Fanuc TP program (LS listing): GST_CLAMSHELL_L1.LS

/PROG  GST_CLAMSHELL_L1
/ATTR
OWNER           = MNEDITOR;
COMMENT         = "BY ROBOTMASTER";
PROG_SIZE       = 0;
CREATE          = DATE 23-01-04  TIME 08:18:11;
MODIFIED        = DATE 23-01-04  TIME 08:18:11;
FILE_NAME       = ;
VERSION         = 0;
LINE_COUNT      = 5014;
MEMORY_SIZE     = 0;
PROTECT         = READ_WRITE;
TCD:  STACK_SIZE        = 0,
      TASK_PRIORITY     = 50,
      TIME_SLICE        = 0,
      BUSY_LAMP_OFF     = 0,
      ABORT_REQUEST     = 0,
      PAUSE_REQUEST     = 0;
DEFAULT_GROUP   = 1,*,*,*,*;
CONTROL_CODE = 00000000 00000000;
/MN
   1: ;
   2: ! Home ;
   3: ;
   4:  UFRAME_NUM = 7 ;
   5:  UTOOL_NUM = 3 ;
   6: ! Jump to specified pass ;
   7: R[215:passLbl] = 100 + R[180:j];
   8: ! Specify last pass ;
   9: IF R[180:j]>1,JMP LBL[8999] ;
  10: IF R[180:j]>0,JMP LBL[R[215:passLbl]] ;
  11:J P[1]  R[225] % FINE ;
  12: ;
  13: ! Path ;
  14: ;
  15:J P[2]  R[225] % FINE ;
  16:L P[3]  R[157] mm/sec CNT100 Offset,PR[24:Rotate_Offset] ;
  17:L P[4]  R[157] mm/sec CNT100 Offset,PR[24:Rotate_Offset] ;
  18: !Pass1 ;
  19: LBL[101:Pass1] ;
  20:L P[5]  R[157] mm/sec FINE Offset,PR[78:Offst_apprch]  ;
  21: WAIT   0.20(sec) ;
  22:L P[5]  R[157] mm/sec CNT100 TA    0.00sec,CALL RUN_LASER_START Offset,PR[25:Start_Offset] ;
  24:L P[6]  R[157] mm/sec CNT100 Offset,PR[24:Rotate_Offset] ;
  25:L P[7]  R[157] mm/sec CNT100 Offset,PR[24:Rotate_Offset] ;
  26:L P[8]  R[157] mm/sec CNT100 Offset,PR[24:Rotate_Offset] ;
  27:L P[9]  R[157] mm/sec CNT100 Offset,PR[24:Rotate_Offset] ;
  28:L P[10]  R[157] mm/sec CNT100 Offset,PR[24:Rotate_Offset] ;
  29:L P[11]  R[157] mm/sec CNT100 Offset,PR[24:Rotate_Offset] ;
  30:L P[12]  R[157] mm/sec CNT100 Offset,PR[24:Rotate_Offset] ;
  31:L P[13]  R[157] mm/sec CNT100 Offset,PR[24:Rotate_Offset] ;
  32:L P[14]  R[157] mm/sec CNT100 Offset,PR[24:Rotate_Offset] ;
  33:L P[15]  R[157] mm/sec CNT100 Offset,PR[24:Rotate_Offset] ;
  34:L P[16]  R[157] mm/sec CNT100 Offset,PR[24:Rotate_Offset] ;
  35:L P[17]  R[157] mm/sec CNT100 Offset,PR[24:Rotate_Offset] ;
  36:L P[18]  R[157] mm/sec CNT100 Offset,PR[24:Rotate_Offset] ;
  37:L P[19]  R[157] mm/sec CNT100 Offset,PR[24:Rotate_Offset] ;
  38:L P[20]  R[157] mm/sec CNT100 Offset,PR[24:Rotate_Offset] ;
  39:L P[21]  R[157] mm/sec CNT100 Offset,PR[24:Rotate_Offset] ;
  40:L P[22]  R[157] mm/sec CNT100 Offset,PR[24:Rotate_Offset] ;
  41:L P[23]  R[157] mm/sec CNT100 Offset,PR[24:Rotate_Offset] ;
  42:L P[24]  R[157] mm/sec CNT100 Offset,PR[24:Rotate_Offset] ;
  43:L P[25]  R[157] mm/sec CNT100 Offset,PR[24:Rotate_Offset] ;
  44:L P[26]  R[157] mm/sec CNT100 Offset,PR[24:Rotate_Offset] ;
  45:L P[27]  R[157] mm/sec CNT100 Offset,PR[24:Rotate_Offset] ;
  46:L P[28]  R[157] mm/sec CNT100 Offset,PR[24:Rotate_Offset] ;
  47:L P[29]  R[157] mm/sec CNT100 Offset,PR[24:Rotate_Offset] ;
  48:L P[30]  R[157] mm/sec CNT100 Offset,PR[24:Rotate_Offset] ;
  49:L P[31]  R[157] mm/sec CNT100 Offset,PR[24:Rotate_Offset] ;
  50:L P[32]  R[157] mm/sec CNT100 Offset,PR[24:Rotate_Offset] ;
  51:L P[33]  R[157] mm/sec CNT100 Offset,PR[24:Rotate_Offset] ;
  52:L P[34]  R[157] mm/sec CNT100 Offset,PR[24:Rotate_Offset] ;
  53:L P[35]  R[157] mm/sec CNT100 Offset,PR[24:Rotate_Offset] ;
  54:L P[36]  R[157] mm/sec CNT100 Offset,PR[24:Rotate_Offset] ;
  55:L P[37]  R[157] mm/sec CNT100 Offset,PR[24:Rotate_Offset] ;
  56:L P[38]  R[157] mm/sec CNT100 Offset,PR[24:Rotate_Offset] ;
  57:L P[39]  R[157] mm/sec CNT100 Offset,PR[24:Rotate_Offset] ;
  58:L P[40]  R[157] mm/sec CNT100 Offset,PR[24:Rotate_Offset] ;
  59:L P[41]  R[157] mm/sec CNT100 Offset,PR[24:Rotate_Offset] ;
  60:L P[42]  R[157] mm/sec CNT100 Offset,PR[24:Rotate_Offset] ;
  61:L P[43]  R[157] mm/sec CNT100 Offset,PR[24:Rotate_Offset] ;
  62:L P[44]  R[157] mm/sec CNT100 Offset,PR[24:Rotate_Offset] ;
  63:L P[45]  R[157] mm/sec CNT100 Offset,PR[24:Rotate_Offset] ;
  64:L P[46]  R[157] mm/sec CNT100 Offset,PR[24:Rotate_Offset] ;
  65:L P[47]  R[157] mm/sec CNT100 Offset,PR[24:Rotate_Offset] ;
  66:L P[48]  R[157] mm/sec CNT100 Offset,PR[24:Rotate_Offset] ;
  67:L P[49]  R[157] mm/sec CNT100 Offset,PR[24:Rotate_Offset] ;
  68:L P[50]  R[157] mm/sec CNT100 Offset,PR[24:Rotate_Offset] ;
  69:L P[51]  R[157] mm/sec CNT100 Offset,PR[24:Rotate_Offset] ;
  70:L P[52]  R[157] mm/sec CNT100 Offset,PR[24:Rotate_Offset] ;
  71:L P[53]  R[157] mm/sec CNT100 Offset,PR[24:Rotate_Offset] ;
  72:L P[54]  R[157] mm/sec CNT100 Offset,PR[24:Rotate_Offset] ;
  73:L P[55]  R[157] mm/sec CNT100 Offset,PR[24:Rotate_Offset] ;
  74:L P[56]  R[157] mm/sec CNT100 Offset,PR[24:Rotate_Offset] ;
  75:L P[57]  R[157] mm/sec CNT100 Offset,PR[24:Rotate_Offset] ;
  76:L P[58]  R[157] mm/sec CNT100 Offset,PR[24:Rotate_Offset] ;
  77:L P[59]  R[157] mm/sec CNT100 TA    0.00sec,CALL RUN_LASER_STOP Offset,PR[26:Stop_Offset] ;
  79:L P[59]  R[157] mm/sec FINE Offset,PR[76:Offst_dprt] ;
  80:L P[60]  R[157] mm/sec CNT100 Offset,PR[24:Rotate_Offset] ;
  81:L P[61]  R[157] mm/sec CNT100 Offset,PR[24:Rotate_Offset] ;
  82:L P[62]  R[157] mm/sec CNT100 Offset,PR[24:Rotate_Offset] ;
  83:L P[63]  R[157] mm/sec CNT100 Offset,PR[24:Rotate_Offset] ;
  84:L P[64]  R[157] mm/sec CNT100 Offset,PR[24:Rotate_Offset] ;
  85:L P[65]  R[157] mm/sec CNT100 Offset,PR[24:Rotate_Offset] ;
  86: !Pass2 ;
  87: LBL[102:Pass2] ;
  88:L P[66]  R[157] mm/sec FINE Offset,PR[78:Offst_apprch]  ;
  89: WAIT   0.20(sec) ;
  90:L P[66]  R[157] mm/sec CNT100 TA    0.00sec,CALL RUN_LASER_START Offset,PR[25:Start_Offset] ;
  92:L P[67]  R[157] mm/sec CNT100 Offset,PR[24:Rotate_Offset] ;
  93:L P[68]  R[157] mm/sec CNT100 Offset,PR[24:Rotate_Offset] ;
  94:L P[69]  R[157] mm/sec CNT100 Offset,PR[24:Rotate_Offset] ;
  95:L P[70]  R[157] mm/sec CNT100 Offset,PR[24:Rotate_Offset] ;
  96:L P[71]  R[157] mm/sec CNT100 Offset,PR[24:Rotate_Offset] ;
  97:L P[72]  R[157] mm/sec CNT100 Offset,PR[24:Rotate_Offset] ;
  98:L P[73]  R[157] mm/sec CNT100 Offset,PR[24:Rotate_Offset] ;
  99:L P[74]  R[157] mm/sec CNT100 Offset,PR[24:Rotate_Offset] ;
 100:L P[75]  R[157] mm/sec CNT100 Offset,PR[24:Rotate_Offset] ;
 101:L P[76]  R[157] mm/sec CNT100 Offset,PR[24:Rotate_Offset] ;
 102:L P[77]  R[157] mm/sec CNT100 Offset,PR[24:Rotate_Offset] ;
 103:L P[78]  R[157] mm/sec CNT100 Offset,PR[24:Rotate_Offset] ;
 104:L P[79]  R[157] mm/sec CNT100 Offset,PR[24:Rotate_Offset] ;
 105:L P[80]  R[157] mm/sec CNT100 Offset,PR[24:Rotate_Offset] ;
 106:L P[81]  R[157] mm/sec CNT100 Offset,PR[24:Rotate_Offset] ;
 107:L P[82]  R[157] mm/sec CNT100 Offset,PR[24:Rotate_Offset] ;
 108:L P[83]  R[157] mm/sec CNT100 Offset,PR[24:Rotate_Offset] ;
 109:L P[84]  R[157] mm/sec CNT100 Offset,PR[24:Rotate_Offset] ;
 110:L P[85]  R[157] mm/sec CNT100 Offset,PR[24:Rotate_Offset] ;
 111:L P[86]  R[157] mm/sec CNT100 Offset,PR[24:Rotate_Offset] ;
 112:L P[87]  R[157] mm/sec CNT100 Offset,PR[24:Rotate_Offset] ;
 113:L P[88]  R[157] mm/sec CNT100 Offset,PR[24:Rotate_Offset] ;
 114:L P[89]  R[157] mm/sec CNT100 Offset,PR[24:Rotate_Offset] ;
 115:L P[90]  R[157] mm/sec CNT100 Offset,PR[24:Rotate_Offset] ;
 116:L P[91]  R[157] mm/sec CNT100 Offset,PR[24:Rotate_Offset] ;
 117:L P[92]  R[157] mm/sec CNT100 Offset,PR[24:Rotate_Offset] ;
 118:L P[93]  R[157] mm/sec CNT100 Offset,PR[24:Rotate_Offset] ;
 119:L P[94]  R[157] mm/sec CNT100 Offset,PR[24:Rotate_Offset] ;
 120:L P[95]  R[157] mm/sec CNT100 Offset,PR[24:Rotate_Offset] ;
 121:L P[96]  R[157] mm/sec CNT100 Offset,PR[24:Rotate_Offset] ;
 122:L P[97]  R[157] mm/sec CNT100 Offset,PR[24:Rotate_Offset] ;
 123:L P[98]  R[157] mm/sec CNT100 Offset,PR[24:Rotate_Offset] ;
 124:L P[99]  R[157] mm/sec CNT100 Offset,PR[24:Rotate_Offset] ;
 125:L P[100]  R[157] mm/sec CNT100 Offset,PR[24:Rotate_Offset] ;
 126:L P[101]  R[157] mm/sec CNT100 Offset,PR[24:Rotate_Offset] ;
 127:L P[102]  R[157] mm/sec CNT100 Offset,PR[24:Rotate_Offset] ;
 128:L P[103]  R[157] mm/sec CNT100 Offset,PR[24:Rotate_Offset] ;
 129:L P[104]  R[157] mm/sec CNT100 Offset,PR[24:Rotate_Offset] ;
 130:L P[105]  R[157] mm/sec CNT100 Offset,PR[24:Rotate_Offset] ;
 131:L P[106]  R[157] mm/sec CNT100 Offset,PR[24:Rotate_Offset] ;
 132:L P[107]  R[157] mm/sec CNT100 Offset,PR[24:Rotate_Offset] ;
 133:L P[108]  R[157] mm/sec CNT100 Offset,PR[24:Rotate_Offset] ;
 134:L P[109]  R[157] mm/sec CNT100 Offset,PR[24:Rotate_Offset] ;
 135:L P[110]  R[157] mm/sec CNT100 Offset,PR[24:Rotate_Offset] ;
 136:L P[111]  R[157] mm/sec CNT100 Offset,PR[24:Rotate_Offset] ;
 137:L P[112]  R[157] mm/sec CNT100 Offset,PR[24:Rotate_Offset] ;
 138:L P[113]  R[157] mm/sec CNT100 Offset,PR[24:Rotate_Offset] ;
 139:L P[114]  R[157] mm/sec CNT100 Offset,PR[24:Rotate_Offset] ;
 140:L P[115]  R[157] mm/sec CNT100 Offset,PR[24:Rotate_Offset] ;
 141:L P[116]  R[157] mm/sec CNT100 Offset,PR[24:Rotate_Offset] ;
 142:L P[117]  R[157] mm/sec CNT100 Offset,PR[24:Rotate_Offset] ;
 143:L P[118]  R[157] mm/sec CNT100 Offset,PR[24:Rotate_Offset] ;
 144:L P[119]  R[157] mm/sec CNT100 Offset,PR[24:Rotate_Offset] ;
 145:L P[120]  R[157] mm/sec CNT100 Offset,PR[24:Rotate_Offset] ;
 146:L P[121]  R[157] mm/sec CNT100 TA    0.00sec,CALL RUN_LASER_STOP Offset,PR[26:Stop_Offset] ;
 148:L P[121]  R[157] mm/sec FINE Offset,PR[76:Offst_dprt] ;
 149:L P[122]  R[157] mm/sec CNT100 Offset,PR[24:Rotate_Offset] ;
 150:L P[123]  R[157] mm/sec CNT100 Offset,PR[24:Rotate_Offset] ;
 151:L P[124]  R[157] mm/sec CNT100 Offset,PR[24:Rotate_Offset] ;
 152:L P[125]  R[157] mm/sec CNT100 Offset,PR[24:Rotate_Offset] ;
 153:L P[126]  R[157] mm/sec CNT100 Offset,PR[24:Rotate_Offset] ;
 154:L P[127]  R[157] mm/sec CNT100 Offset,PR[24:Rotate_Offset] ;
 155: !Pass3 ;
 156: LBL[103:Pass3] ;
 157:L P[128]  R[157] mm/sec FINE Offset,PR[78:Offst_apprch]  ;
 158: WAIT   0.20(sec) ;
 159:L P[128]  R[157] mm/sec CNT100 TA    0.00sec,CALL RUN_LASER_START Offset,PR[25:Start_Offset] ;
 161:L P[129]  R[157] mm/sec CNT100 Offset,PR[24:Rotate_Offset] ;
 162:L P[130]  R[157] mm/sec CNT100 Offset,PR[24:Rotate_Offset] ;
 163:L P[131]  R[157] mm/sec CNT100 Offset,PR[24:Rotate_Offset] ;
 164:L P[132]  R[157] mm/sec CNT100 Offset,PR[24:Rotate_Offset] ;
 165:L P[133]  R[157] mm/sec CNT100 Offset,PR[24:Rotate_Offset] ;
 166:L P[134]  R[157] mm/sec CNT100 Offset,PR[24:Rotate_Offset] ;
 167:L P[135]  R[157] mm/sec CNT100 Offset,PR[24:Rotate_Offset] ;
 168:L P[136]  R[157] mm/sec CNT100 Offset,PR[24:Rotate_Offset] ;
 169:L P[137]  R[157] mm/sec CNT100 Offset,PR[24:Rotate_Offset] ;
 170:L P[138]  R[157] mm/sec CNT100 Offset,PR[24:Rotate_Offset] ;
 171:L P[139]  R[157] mm/sec CNT100 Offset,PR[24:Rotate_Offset] ;
 172:L P[140]  R[157] mm/sec CNT100 Offset,PR[24:Rotate_Offset] ;
 173:L P[141]  R[157] mm/sec CNT100 Offset,PR[24:Rotate_Offset] ;
 174:L P[142]  R[157] mm/sec CNT100 Offset,PR[24:Rotate_Offset] ;
 175:L P[143]  R[157] mm/sec CNT100 Offset,PR[24:Rotate_Offset] ;
 176:L P[144]  R[157] mm/sec CNT100 Offset,PR[24:Rotate_Offset] ;
 177:L P[145]  R[157] mm/sec CNT100 Offset,PR[24:Rotate_Offset] ;
 178:L P[146]  R[157] mm/sec CNT100 Offset,PR[24:Rotate_Offset] ;
 179:L P[147]  R[157] mm/sec CNT100 Offset,PR[24:Rotate_Offset] ;
 180:L P[148]  R[157] mm/sec CNT100 Offset,PR[24:Rotate_Offset] ;
 181:L P[149]  R[157] mm/sec CNT100 Offset,PR[24:Rotate_Offset] ;
 182:L P[150]  R[157] mm/sec CNT100 Offset,PR[24:Rotate_Offset] ;
 183:L P[151]  R[157] mm/sec CNT100 Offset,PR[24:Rotate_Offset] ;
 184:L P[152]  R[157] mm/sec CNT100 Offset,PR[24:Rotate_Offset] ;
 185:L P[153]  R[157] mm/sec CNT100 Offset,PR[24:Rotate_Offset] ;
 186:L P[154]  R[157] mm/sec CNT100 Offset,PR[24:Rotate_Offset] ;
 187:L P[155]  R[157] mm/sec CNT100 Offset,PR[24:Rotate_Offset] ;
 188:L P[156]  R[157] mm/sec CNT100 Offset,PR[24:Rotate_Offset] ;
 189:L P[157]  R[157] mm/sec CNT100 Offset,PR[24:Rotate_Offset] ;
 190:L P[158]  R[157] mm/sec CNT100 Offset,PR[24:Rotate_Offset] ;
 191:L P[159]  R[157] mm/sec CNT100 Offset,PR[24:Rotate_Offset] ;
 192:L P[160]  R[157] mm/sec CNT100 Offset,PR[24:Rotate_Offset] ;
 193:L P[161]  R[157] mm/sec CNT100 Offset,PR[24:Rotate_Offset] ;
 194:L P[162]  R[157] mm/sec CNT100 Offset,PR[24:Rotate_Offset] ;
 195:L P[163]  R[157] mm/sec CNT100 Offset,PR[24:Rotate_Offset] ;
 196:L P[164]  R[157] mm/sec CNT100 Offset,PR[24:Rotate_Offset] ;
 197:L P[165]  R[157] mm/sec CNT100 Offset,PR[24:Rotate_Offset] ;
 198:L P[166]  R[157] mm/sec CNT100 Offset,PR[24:Rotate_Offset] ;
 199:L P[167]  R[157] mm/sec CNT100 Offset,PR[24:Rotate_Offset] ;
 200:L P[168]  R[157] mm/sec CNT100 Offset,PR[24:Rotate_Offset] ;
 201:L P[169]  R[157] mm/sec CNT100 Offset,PR[24:Rotate_Offset] ;
 202:L P[170]  R[157] mm/sec CNT100 Offset,PR[24:Rotate_Offset] ;
 203:L P[171]  R[157] mm/sec CNT100 Offset,PR[24:Rotate_Offset] ;
 204:L P[172]  R[157] mm/sec CNT100 Offset,PR[24:Rotate_Offset] ;
 205:L P[173]  R[157] mm/sec CNT100 Offset,PR[24:Rotate_Offset] ;
 206:L P[174]  R[157] mm/sec CNT100 Offset,PR[24:Rotate_Offset] ;
 207:L P[175]  R[157] mm/sec CNT100 Offset,PR[24:Rotate_Offset] ;
 208:L P[176]  R[157] mm/sec CNT100 Offset,PR[24:Rotate_Offset] ;
 209:L P[177]  R[157] mm/sec CNT100 Offset,PR[24:Rotate_Offset] ;
 210:L P[178]  R[157] mm/sec CNT100 Offset,PR[24:Rotate_Offset] ;
 211:L P[179]  R[157] mm/sec CNT100 Offset,PR[24:Rotate_Offset] ;
 212:L P[180]  R[157] mm/sec CNT100 Offset,PR[24:Rotate_Offset] ;
 213:L P[181]  R[157] mm/sec CNT100 Offset,PR[24:Rotate_Offset] ;
 214:L P[182]  R[157] mm/sec CNT100 Offset,PR[24:Rotate_Offset] ;
 215:L P[183]  R[157] mm/sec CNT100 TA    0.00sec,CALL RUN_LASER_STOP Offset,PR[26:Stop_Offset] ;
 217:L P[183]  R[157] mm/sec FINE Offset,PR[76:Offst_dprt] ;
 218:L P[184]  R[157] mm/sec CNT100 Offset,PR[24:Rotate_Offset] ;
 219:L P[185]  R[157] mm/sec CNT100 Offset,PR[24:Rotate_Offset] ;
 220:L P[186]  R[157] mm/sec CNT100 Offset,PR[24:Rotate_Offset] ;
 221:L P[187]  R[157] mm/sec CNT100 Offset,PR[24:Rotate_Offset] ;
 222:L P[188]  R[157] mm/sec CNT100 Offset,PR[24:Rotate_Offset] ;
 223:L P[189]  R[157] mm/sec CNT100 Offset,PR[24:Rotate_Offset] ;
 224: !Pass4 ;
 225: LBL[104:Pass4] ;
 226:L P[190]  R[157] mm/sec FINE Offset,PR[78:Offst_apprch]  ;
 227: WAIT   0.20(sec) ;
 228:L P[190]  R[157] mm/sec CNT100 TA    0.00sec,CALL RUN_LASER_START Offset,PR[25:Start_Offset] ;
 230:L P[191]  R[157] mm/sec CNT100 Offset,PR[24:Rotate_Offset] ;
 231:L P[192]  R[157] mm/sec CNT100 Offset,PR[24:Rotate_Offset] ;
 232:L P[193]  R[157] mm/sec CNT100 Offset,PR[24:Rotate_Offset] ;
 233:L P[194]  R[157] mm/sec CNT100 Offset,PR[24:Rotate_Offset] ;
 234:L P[195]  R[157] mm/sec CNT100 Offset,PR[24:Rotate_Offset] ;
 235:L P[196]  R[157] mm/sec CNT100 Offset,PR[24:Rotate_Offset] ;
 236:L P[197]  R[157] mm/sec CNT100 Offset,PR[24:Rotate_Offset] ;
 237:L P[198]  R[157] mm/sec CNT100 Offset,PR[24:Rotate_Offset] ;
 238:L P[199]  R[157] mm/sec CNT100 Offset,PR[24:Rotate_Offset] ;
 239:L P[200]  R[157] mm/sec CNT100 Offset,PR[24:Rotate_Offset] ;
 240:L P[201]  R[157] mm/sec CNT100 Offset,PR[24:Rotate_Offset] ;
 241:L P[202]  R[157] mm/sec CNT100 Offset,PR[24:Rotate_Offset] ;
 242:L P[203]  R[157] mm/sec CNT100 Offset,PR[24:Rotate_Offset] ;
 243:L P[204]  R[157] mm/sec CNT100 Offset,PR[24:Rotate_Offset] ;
 244:L P[205]  R[157] mm/sec CNT100 Offset,PR[24:Rotate_Offset] ;
 245:L P[206]  R[157] mm/sec CNT100 Offset,PR[24:Rotate_Offset] ;
 246:L P[207]  R[157] mm/sec CNT100 Offset,PR[24:Rotate_Offset] ;
 247:L P[208]  R[157] mm/sec CNT100 Offset,PR[24:Rotate_Offset] ;
 248:L P[209]  R[157] mm/sec CNT100 Offset,PR[24:Rotate_Offset] ;
 249:L P[210]  R[157] mm/sec CNT100 Offset,PR[24:Rotate_Offset] ;
 250:L P[211]  R[157] mm/sec CNT100 Offset,PR[24:Rotate_Offset] ;
 251:L P[212]  R[157] mm/sec CNT100 Offset,PR[24:Rotate_Offset] ;
 252:L P[213]  R[157] mm/sec CNT100 Offset,PR[24:Rotate_Offset] ;
 253:L P[214]  R[157] mm/sec CNT100 Offset,PR[24:Rotate_Offset] ;
 254:L P[215]  R[157] mm/sec CNT100 Offset,PR[24:Rotate_Offset] ;
 255:L P[216]  R[157] mm/sec CNT100 Offset,PR[24:Rotate_Offset] ;
 256:L P[217]  R[157] mm/sec CNT100 Offset,PR[24:Rotate_Offset] ;
 257:L P[218]  R[157] mm/sec CNT100 Offset,PR[24:Rotate_Offset] ;
 258:L P[219]  R[157] mm/sec CNT100 Offset,PR[24:Rotate_Offset] ;
 259:L P[220]  R[157] mm/sec CNT100 Offset,PR[24:Rotate_Offset] ;
 260:L P[221]  R[157] mm/sec CNT100 Offset,PR[24:Rotate_Offset] ;
 261:L P[222]  R[157] mm/sec CNT100 Offset,PR[24:Rotate_Offset] ;
 262:L P[223]  R[157] mm/sec CNT100 Offset,PR[24:Rotate_Offset] ;
 263:L P[224]  R[157] mm/sec CNT100 Offset,PR[24:Rotate_Offset] ;
 264:L P[225]  R[157] mm/sec CNT100 Offset,PR[24:Rotate_Offset] ;
 265:L P[226]  R[157] mm/sec CNT100 Offset,PR[24:Rotate_Offset] ;
 266:L P[227]  R[157] mm/sec CNT100 Offset,PR[24:Rotate_Offset] ;
 267:L P[228]  R[157] mm/sec CNT100 Offset,PR[24:Rotate_Offset] ;
 268:L P[229]  R[157] mm/sec CNT100 Offset,PR[24:Rotate_Offset] ;
 269:L P[230]  R[157] mm/sec CNT100 Offset,PR[24:Rotate_Offset] ;
 270:L P[231]  R[157] mm/sec CNT100 Offset,PR[24:Rotate_Offset] ;
 271:L P[232]  R[157] mm/sec CNT100 Offset,PR[24:Rotate_Offset] ;
 272:L P[233]  R[157] mm/sec CNT100 Offset,PR[24:Rotate_Offset] ;
 273:L P[234]  R[157] mm/sec CNT100 Offset,PR[24:Rotate_Offset] ;
 274:L P[235]  R[157] mm/sec CNT100 Offset,PR[24:Rotate_Offset] ;
 275:L P[236]  R[157] mm/sec CNT100 Offset,PR[24:Rotate_Offset] ;
 276:L P[237]  R[157] mm/sec CNT100 Offset,PR[24:Rotate_Offset] ;
 277:L P[238]  R[157] mm/sec CNT100 TA    0.00sec,CALL RUN_LASER_STOP Offset,PR[26:Stop_Offset] ;
 279:L P[238]  R[157] mm/sec FINE Offset,PR[76:Offst_dprt] ;
 280:L P[239]  R[157] mm/sec CNT100 Offset,PR[24:Rotate_Offset] ;
 281:L P[240]  R[157] mm/sec CNT100 Offset,PR[24:Rotate_Offset] ;
 282:L P[241]  R[157] mm/sec CNT100 Offset,PR[24:Rotate_Offset] ;
 283:L P[242]  R[157] mm/sec CNT100 Offset,PR[24:Rotate_Offset] ;
 284:L P[243]  R[157] mm/sec CNT100 Offset,PR[24:Rotate_Offset] ;
 285:L P[244]  R[157] mm/sec CNT100 Offset,PR[24:Rotate_Offset] ;
 286: !Pass5 ;
 287: LBL[105:Pass5] ;
 288:L P[245]  R[157] mm/sec FINE Offset,PR[78:Offst_apprch]  ;
 289: WAIT   0.20(sec) ;
 290:L P[245]  R[157] mm/sec CNT100 TA    0.00sec,CALL RUN_LASER_START Offset,PR[25:Start_Offset] ;
 292:L P[246]  R[157] mm/sec CNT100 Offset,PR[24:Rotate_Offset] ;
 293:L P[247]  R[157] mm/sec CNT100 Offset,PR[24:Rotate_Offset] ;
 294:L P[248]  R[157] mm/sec CNT100 Offset,PR[24:Rotate_Offset] ;
 295:L P[249]  R[157] mm/sec CNT100 Offset,PR[24:Rotate_Offset] ;
 296:L P[250]  R[157] mm/sec CNT100 Offset,PR[24:Rotate_Offset] ;
 297:L P[251]  R[157] mm/sec CNT100 Offset,PR[24:Rotate_Offset] ;
 298:L P[252]  R[157] mm/sec CNT100 Offset,PR[24:Rotate_Offset] ;
 299:L P[253]  R[157] mm/sec CNT100 Offset,PR[24:Rotate_Offset] ;
 300:L P[254]  R[157] mm/sec CNT100 Offset,PR[24:Rotate_Offset] ;
 301:L P[255]  R[157] mm/sec CNT100 Offset,PR[24:Rotate_Offset] ;
 302:L P[256]  R[157] mm/sec CNT100 Offset,PR[24:Rotate_Offset] ;
 303:L P[257]  R[157] mm/sec CNT100 Offset,PR[24:Rotate_Offset] ;
 304:L P[258]  R[157] mm/sec CNT100 Offset,PR[24:Rotate_Offset] ;
 305:L P[259]  R[157] mm/sec CNT100 Offset,PR[24:Rotate_Offset] ;
 306:L P[260]  R[157] mm/sec CNT100 Offset,PR[24:Rotate_Offset] ;
 307:L P[261]  R[157] mm/sec CNT100 Offset,PR[24:Rotate_Offset] ;
 308:L P[262]  R[157] mm/sec CNT100 Offset,PR[24:Rotate_Offset] ;
 309:L P[263]  R[157] mm/sec CNT100 Offset,PR[24:Rotate_Offset] ;
 310:L P[264]  R[157] mm/sec CNT100 Offset,PR[24:Rotate_Offset] ;
 311:L P[265]  R[157] mm/sec CNT100 Offset,PR[24:Rotate_Offset] ;
 312:L P[266]  R[157] mm/sec CNT100 Offset,PR[24:Rotate_Offset] ;
 313:L P[267]  R[157] mm/sec CNT100 Offset,PR[24:Rotate_Offset] ;
 314:L P[268]  R[157] mm/sec CNT100 Offset,PR[24:Rotate_Offset] ;
 315:L P[269]  R[157] mm/sec CNT100 Offset,PR[24:Rotate_Offset] ;
 316:L P[270]  R[157] mm/sec CNT100 Offset,PR[24:Rotate_Offset] ;
 317:L P[271]  R[157] mm/sec CNT100 Offset,PR[24:Rotate_Offset] ;
 318:L P[272]  R[157] mm/sec CNT100 Offset,PR[24:Rotate_Offset] ;
 319:L P[273]  R[157] mm/sec CNT100 Offset,PR[24:Rotate_Offset] ;
 320:L P[274]  R[157] mm/sec CNT100 Offset,PR[24:Rotate_Offset] ;
 321:L P[275]  R[157] mm/sec CNT100 Offset,PR[24:Rotate_Offset] ;
 322:L P[276]  R[157] mm/sec CNT100 Offset,PR[24:Rotate_Offset] ;
 323:L P[277]  R[157] mm/sec CNT100 Offset,PR[24:Rotate_Offset] ;
 324:L P[278]  R[157] mm/sec CNT100 Offset,PR[24:Rotate_Offset] ;
 325:L P[279]  R[157] mm/sec CNT100 Offset,PR[24:Rotate_Offset] ;
 326:L P[280]  R[157] mm/sec CNT100 Offset,PR[24:Rotate_Offset] ;
 327:L P[281]  R[157] mm/sec CNT100 Offset,PR[24:Rotate_Offset] ;
 328:L P[282]  R[157] mm/sec CNT100 Offset,PR[24:Rotate_Offset] ;
 329:L P[283]  R[157] mm/sec CNT100 Offset,PR[24:Rotate_Offset] ;
 330:L P[284]  R[157] mm/sec CNT100 Offset,PR[24:Rotate_Offset] ;
 331:L P[285]  R[157] mm/sec CNT100 Offset,PR[24:Rotate_Offset] ;
 332:L P[286]  R[157] mm/sec CNT100 Offset,PR[24:Rotate_Offset] ;
 333:L P[287]  R[157] mm/sec CNT100 Offset,PR[24:Rotate_Offset] ;
 334:L P[288]  R[157] mm/sec CNT100 Offset,PR[24:Rotate_Offset] ;
 335:L P[289]  R[157] mm/sec CNT100 Offset,PR[24:Rotate_Offset] ;
 336:L P[290]  R[157] mm/sec CNT100 Offset,PR[24:Rotate_Offset] ;
 337:L P[291]  R[157] mm/sec CNT100 Offset,PR[24:Rotate_Offset] ;
 338:L P[292]  R[157] mm/sec CNT100 Offset,PR[24:Rotate_Offset] ;
 339:L P[293]  R[157] mm/sec CNT100 TA    0.00sec,CALL RUN_LASER_STOP Offset,PR[26:Stop_Offset] ;
 341:L P[293]  R[157] mm/sec FINE Offset,PR[76:Offst_dprt] ;
 342:L P[294]  R[157] mm/sec CNT100 Offset,PR[24:Rotate_Offset] ;
 343:L P[295]  R[157] mm/sec CNT100 Offset,PR[24:Rotate_Offset] ;
 344:L P[296]  R[157] mm/sec CNT100 Offset,PR[24:Rotate_Offset] ;
 345:L P[297]  R[157] mm/sec CNT100 Offset,PR[24:Rotate_Offset] ;
 346:L P[298]  R[157] mm/sec CNT100 Offset,PR[24:Rotate_Offset] ;
 347:L P[299]  R[157] mm/sec CNT100 Offset,PR[24:Rotate_Offset] ;
 348: !Pass6 ;
 349: LBL[106:Pass6] ;
 350:L P[300]  R[157] mm/sec FINE Offset,PR[78:Offst_apprch]  ;
 351: WAIT   0.20(sec) ;
 352:L P[300]  R[157] mm/sec CNT100 TA    0.00sec,CALL RUN_LASER_START Offset,PR[25:Start_Offset] ;
 354:L P[301]  R[157] mm/sec CNT100 Offset,PR[24:Rotate_Offset] ;
 355:L P[302]  R[157] mm/sec CNT100 Offset,PR[24:Rotate_Offset] ;
 356:L P[303]  R[157] mm/sec CNT100 Offset,PR[24:Rotate_Offset] ;
 357:L P[304]  R[157] mm/sec CNT100 Offset,PR[24:Rotate_Offset] ;
 358:L P[305]  R[157] mm/sec CNT100 Offset,PR[24:Rotate_Offset] ;
 359:L P[306]  R[157] mm/sec CNT100 Offset,PR[24:Rotate_Offset] ;
 360:L P[307]  R[157] mm/sec CNT100 Offset,PR[24:Rotate_Offset] ;
 361:L P[308]  R[157] mm/sec CNT100 Offset,PR[24:Rotate_Offset] ;
 362:L P[309]  R[157] mm/sec CNT100 Offset,PR[24:Rotate_Offset] ;
 363:L P[310]  R[157] mm/sec CNT100 Offset,PR[24:Rotate_Offset] ;
 364:L P[311]  R[157] mm/sec CNT100 Offset,PR[24:Rotate_Offset] ;
 365:L P[312]  R[157] mm/sec CNT100 Offset,PR[24:Rotate_Offset] ;
 366:L P[313]  R[157] mm/sec CNT100 Offset,PR[24:Rotate_Offset] ;
 367:L P[314]  R[157] mm/sec CNT100 Offset,PR[24:Rotate_Offset] ;
 368:L P[315]  R[157] mm/sec CNT100 Offset,PR[24:Rotate_Offset] ;
 369:L P[316]  R[157] mm/sec CNT100 Offset,PR[24:Rotate_Offset] ;
 370:L P[317]  R[157] mm/sec CNT100 Offset,PR[24:Rotate_Offset] ;
 371:L P[318]  R[157] mm/sec CNT100 Offset,PR[24:Rotate_Offset] ;
 372:L P[319]  R[157] mm/sec CNT100 Offset,PR[24:Rotate_Offset] ;
 373:L P[320]  R[157] mm/sec CNT100 Offset,PR[24:Rotate_Offset] ;
 374:L P[321]  R[157] mm/sec CNT100 Offset,PR[24:Rotate_Offset] ;
 375:L P[322]  R[157] mm/sec CNT100 Offset,PR[24:Rotate_Offset] ;
 376:L P[323]  R[157] mm/sec CNT100 Offset,PR[24:Rotate_Offset] ;
 377:L P[324]  R[157] mm/sec CNT100 Offset,PR[24:Rotate_Offset] ;
 378:L P[325]  R[157] mm/sec CNT100 Offset,PR[24:Rotate_Offset] ;
 379:L P[326]  R[157] mm/sec CNT100 Offset,PR[24:Rotate_Offset] ;
 380:L P[327]  R[157] mm/sec CNT100 Offset,PR[24:Rotate_Offset] ;
 381:L P[328]  R[157] mm/sec CNT100 Offset,PR[24:Rotate_Offset] ;
 382:L P[329]  R[157] mm/sec CNT100 Offset,PR[24:Rotate_Offset] ;
 383:L P[330]  R[157] mm/sec CNT100 Offset,PR[24:Rotate_Offset] ;
 384:L P[331]  R[157] mm/sec CNT100 Offset,PR[24:Rotate_Offset] ;
 385:L P[332]  R[157] mm/sec CNT100 Offset,PR[24:Rotate_Offset] ;
 386:L P[333]  R[157] mm/sec CNT100 Offset,PR[24:Rotate_Offset] ;
 387:L P[334]  R[157] mm/sec CNT100 Offset,PR[24:Rotate_Offset] ;
 388:L P[335]  R[157] mm/sec CNT100 Offset,PR[24:Rotate_Offset] ;
 389:L P[336]  R[157] mm/sec CNT100 Offset,PR[24:Rotate_Offset] ;
 390:L P[337]  R[157] mm/sec CNT100 Offset,PR[24:Rotate_Offset] ;
 391:L P[338]  R[157] mm/sec CNT100 Offset,PR[24:Rotate_Offset] ;
 392:L P[339]  R[157] mm/sec CNT100 Offset,PR[24:Rotate_Offset] ;
 393:L P[340]  R[157] mm/sec CNT100 Offset,PR[24:Rotate_Offset] ;
 394:L P[341]  R[157] mm/sec CNT100 Offset,PR[24:Rotate_Offset] ;
 395:L P[342]  R[157] mm/sec CNT100 Offset,PR[24:Rotate_Offset] ;
 396:L P[343]  R[157] mm/sec CNT100 Offset,PR[24:Rotate_Offset] ;
 397:L P[344]  R[157] mm/sec CNT100 Offset,PR[24:Rotate_Offset] ;
 398:L P[345]  R[157] mm/sec CNT100 Offset,PR[24:Rotate_Offset] ;
 399:L P[346]  R[157] mm/sec CNT100 Offset,PR[24:Rotate_Offset] ;
 400:L P[347]  R[157] mm/sec CNT100 Offset,PR[24:Rotate_Offset] ;
 401:L P[348]  R[157] mm/sec CNT100 TA    0.00sec,CALL RUN_LASER_STOP Offset,PR[26:Stop_Offset] ;
 403:L P[348]  R[157] mm/sec FINE Offset,PR[76:Offst_dprt] ;
 404:L P[349]  R[157] mm/sec CNT100 Offset,PR[24:Rotate_Offset] ;
 405:L P[350]  R[157] mm/sec CNT100 Offset,PR[24:Rotate_Offset] ;
 406:L P[351]  R[157] mm/sec CNT100 Offset,PR[24:Rotate_Offset] ;
 407:L P[352]  R[157] mm/sec CNT100 Offset,PR[24:Rotate_Offset] ;
 408:L P[353]  R[157] mm/sec CNT100 Offset,PR[24:Rotate_Offset] ;
 409:L P[354]  R[157] mm/sec CNT100 Offset,PR[24:Rotate_Offset] ;
 410: !Pass7 ;
 411: LBL[107:Pass7] ;
 412:L P[355]  R[157] mm/sec FINE Offset,PR[78:Offst_apprch]  ;
 413: WAIT   0.20(sec) ;
 414:L P[355]  R[157] mm/sec CNT100 TA    0.00sec,CALL RUN_LASER_START Offset,PR[25:Start_Offset] ;
 416:L P[356]  R[157] mm/sec CNT100 Offset,PR[24:Rotate_Offset] ;
 417:L P[357]  R[157] mm/sec CNT100 Offset,PR[24:Rotate_Offset] ;
 418:L P[358]  R[157] mm/sec CNT100 Offset,PR[24:Rotate_Offset] ;
 419:L P[359]  R[157] mm/sec CNT100 Offset,PR[24:Rotate_Offset] ;
 420:L P[360]  R[157] mm/sec CNT100 Offset,PR[24:Rotate_Offset] ;
 421:L P[361]  R[157] mm/sec CNT100 Offset,PR[24:Rotate_Offset] ;
 422:L P[362]  R[157] mm/sec CNT100 Offset,PR[24:Rotate_Offset] ;
 423:L P[363]  R[157] mm/sec CNT100 TA    0.00sec,CALL RUN_LASER_STOP Offset,PR[26:Stop_Offset] ;
 425:L P[363]  R[157] mm/sec FINE Offset,PR[76:Offst_dprt] ;
 426:L P[364]  R[157] mm/sec CNT100 Offset,PR[24:Rotate_Offset] ;
 427:L P[365]  R[157] mm/sec CNT100 Offset,PR[24:Rotate_Offset] ;
 428:L P[366]  R[157] mm/sec CNT100 Offset,PR[24:Rotate_Offset] ;
 429:L P[367]  R[157] mm/sec CNT100 Offset,PR[24:Rotate_Offset] ;
 430:L P[368]  R[157] mm/sec CNT100 Offset,PR[24:Rotate_Offset] ;
 431:L P[369]  R[157] mm/sec CNT100 Offset,PR[24:Rotate_Offset] ;
 432: !Pass8 ;
 433: LBL[108:Pass8] ;
 434:L P[370]  R[157] mm/sec FINE Offset,PR[78:Offst_apprch]  ;
 435: WAIT   0.20(sec) ;
 436:L P[370]  R[157] mm/sec CNT100 TA    0.00sec,CALL RUN_LASER_START Offset,PR[25:Start_Offset] ;
 438:L P[371]  R[157] mm/sec CNT100 Offset,PR[24:Rotate_Offset] ;
 439:L P[372]  R[157] mm/sec CNT100 Offset,PR[24:Rotate_Offset] ;
 440:L P[373]  R[157] mm/sec CNT100 Offset,PR[24:Rotate_Offset] ;
 441:L P[374]  R[157] mm/sec CNT100 Offset,PR[24:Rotate_Offset] ;
 442:L P[375]  R[157] mm/sec CNT100 Offset,PR[24:Rotate_Offset] ;
 443:L P[376]  R[157] mm/sec CNT100 Offset,PR[24:Rotate_Offset] ;
 444:L P[377]  R[157] mm/sec CNT100 Offset,PR[24:Rotate_Offset] ;
 445:L P[378]  R[157] mm/sec CNT100 Offset,PR[24:Rotate_Offset] ;
 446:L P[379]  R[157] mm/sec CNT100 Offset,PR[24:Rotate_Offset] ;
 447:L P[380]  R[157] mm/sec CNT100 Offset,PR[24:Rotate_Offset] ;
 448:L P[381]  R[157] mm/sec CNT100 Offset,PR[24:Rotate_Offset] ;
 449:L P[382]  R[157] mm/sec CNT100 Offset,PR[24:Rotate_Offset] ;
 450:L P[383]  R[157] mm/sec CNT100 Offset,PR[24:Rotate_Offset] ;
 451:L P[384]  R[157] mm/sec CNT100 Offset,PR[24:Rotate_Offset] ;
 452:L P[385]  R[157] mm/sec CNT100 Offset,PR[24:Rotate_Offset] ;
 453:L P[386]  R[157] mm/sec CNT100 Offset,PR[24:Rotate_Offset] ;
 454:L P[387]  R[157] mm/sec CNT100 Offset,PR[24:Rotate_Offset] ;
 455:L P[388]  R[157] mm/sec CNT100 Offset,PR[24:Rotate_Offset] ;
 456:L P[389]  R[157] mm/sec CNT100 TA    0.00sec,CALL RUN_LASER_STOP Offset,PR[26:Stop_Offset] ;
 458:L P[389]  R[157] mm/sec FINE Offset,PR[76:Offst_dprt] ;
 459:L P[390]  R[157] mm/sec CNT100 Offset,PR[24:Rotate_Offset] ;
 460:L P[391]  R[157] mm/sec CNT100 Offset,PR[24:Rotate_Offset] ;
 461:L P[392]  R[157] mm/sec CNT100 Offset,PR[24:Rotate_Offset] ;
 462:L P[393]  R[157] mm/sec CNT100 Offset,PR[24:Rotate_Offset] ;
 463:L P[394]  R[157] mm/sec CNT100 Offset,PR[24:Rotate_Offset] ;
 464:L P[395]  R[157] mm/sec CNT100 Offset,PR[24:Rotate_Offset] ;
 465: !Pass9 ;
 466: LBL[109:Pass9] ;
 467:L P[396]  R[157] mm/sec FINE Offset,PR[78:Offst_apprch]  ;
 468: WAIT   0.20(sec) ;
 469:L P[396]  R[157] mm/sec CNT100 TA    0.00sec,CALL RUN_LASER_START Offset,PR[25:Start_Offset] ;
 471:L P[397]  R[157] mm/sec CNT100 Offset,PR[24:Rotate_Offset] ;
 472:L P[398]  R[157] mm/sec CNT100 Offset,PR[24:Rotate_Offset] ;
 473:L P[399]  R[157] mm/sec CNT100 Offset,PR[24:Rotate_Offset] ;
 474:L P[400]  R[157] mm/sec CNT100 Offset,PR[24:Rotate_Offset] ;
 475:L P[401]  R[157] mm/sec CNT100 Offset,PR[24:Rotate_Offset] ;
 476:L P[402]  R[157] mm/sec CNT100 Offset,PR[24:Rotate_Offset] ;
 477:L P[403]  R[157] mm/sec CNT100 TA    0.00sec,CALL RUN_LASER_STOP Offset,PR[26:Stop_Offset] ;
 479:L P[403]  R[157] mm/sec FINE Offset,PR[76:Offst_dprt] ;
 480:L P[404]  R[157] mm/sec CNT100 Offset,PR[24:Rotate_Offset] ;
 481:L P[405]  R[157] mm/sec CNT100 Offset,PR[24:Rotate_Offset] ;
 482:L P[406]  R[157] mm/sec CNT100 Offset,PR[24:Rotate_Offset] ;
 483:L P[407]  R[157] mm/sec CNT100 Offset,PR[24:Rotate_Offset] ;
 484:L P[408]  R[157] mm/sec CNT100 Offset,PR[24:Rotate_Offset] ;
 485:L P[409]  R[157] mm/sec CNT100 Offset,PR[24:Rotate_Offset] ;
 486: !Pass10 ;
 487: LBL[110:Pass10] ;
 488:L P[410]  R[157] mm/sec FINE Offset,PR[78:Offst_apprch]  ;
 489: WAIT   0.20(sec) ;
 490:L P[410]  R[157] mm/sec CNT100 TA    0.00sec,CALL RUN_LASER_START Offset,PR[25:Start_Offset] ;
 492:L P[411]  R[157] mm/sec CNT100 Offset,PR[24:Rotate_Offset] ;
 493:L P[412]  R[157] mm/sec CNT100 Offset,PR[24:Rotate_Offset] ;
 494:L P[413]  R[157] mm/sec CNT100 Offset,PR[24:Rotate_Offset] ;
 495:L P[414]  R[157] mm/sec CNT100 Offset,PR[24:Rotate_Offset] ;
 496:L P[415]  R[157] mm/sec CNT100 Offset,PR[24:Rotate_Offset] ;
 497:L P[416]  R[157] mm/sec CNT100 Offset,PR[24:Rotate_Offset] ;
 498:L P[417]  R[157] mm/sec CNT100 Offset,PR[24:Rotate_Offset] ;
 499:L P[418]  R[157] mm/sec CNT100 Offset,PR[24:Rotate_Offset] ;
 500:L P[419]  R[157] mm/sec CNT100 Offset,PR[24:Rotate_Offset] ;
 501:L P[420]  R[157] mm/sec CNT100 Offset,PR[24:Rotate_Offset] ;
 502:L P[421]  R[157] mm/sec CNT100 Offset,PR[24:Rotate_Offset] ;
 503:L P[422]  R[157] mm/sec CNT100 Offset,PR[24:Rotate_Offset] ;
 504:L P[423]  R[157] mm/sec CNT100 Offset,PR[24:Rotate_Offset] ;
 505:L P[424]  R[157] mm/sec CNT100 TA    0.00sec,CALL RUN_LASER_STOP Offset,PR[26:Stop_Offset] ;
 507:L P[424]  R[157] mm/sec FINE Offset,PR[76:Offst_dprt] ;
 508:L P[425]  R[157] mm/sec CNT100 Offset,PR[24:Rotate_Offset] ;
 509:L P[426]  R[157] mm/sec CNT100 Offset,PR[24:Rotate_Offset] ;
 510:L P[427]  R[157] mm/sec CNT100 Offset,PR[24:Rotate_Offset] ;
 511:L P[428]  R[157] mm/sec CNT100 Offset,PR[24:Rotate_Offset] ;
 512:L P[429]  R[157] mm/sec CNT100 Offset,PR[24:Rotate_Offset] ;
 513:L P[430]  R[157] mm/sec CNT100 Offset,PR[24:Rotate_Offset] ;
 514: !Pass11 ;
 515: LBL[111:Pass11] ;
 516:L P[431]  R[157] mm/sec FINE Offset,PR[78:Offst_apprch]  ;
 517: WAIT   0.20(sec) ;
 518:L P[431]  R[157] mm/sec CNT100 TA    0.00sec,CALL RUN_LASER_START Offset,PR[25:Start_Offset] ;
 520:L P[432]  R[157] mm/sec CNT100 Offset,PR[24:Rotate_Offset] ;
 521:L P[433]  R[157] mm/sec CNT100 Offset,PR[24:Rotate_Offset] ;
 522:L P[434]  R[157] mm/sec CNT100 Offset,PR[24:Rotate_Offset] ;
 523:L P[435]  R[157] mm/sec CNT100 Offset,PR[24:Rotate_Offset] ;
 524:L P[436]  R[157] mm/sec CNT100 Offset,PR[24:Rotate_Offset] ;
 525:L P[437]  R[157] mm/sec CNT100 Offset,PR[24:Rotate_Offset] ;
 526:L P[438]  R[157] mm/sec CNT100 TA    0.00sec,CALL RUN_LASER_STOP Offset,PR[26:Stop_Offset] ;
 528:L P[438]  R[157] mm/sec FINE Offset,PR[76:Offst_dprt] ;
 529:L P[439]  R[157] mm/sec CNT100 Offset,PR[24:Rotate_Offset] ;
 530:L P[440]  R[157] mm/sec CNT100 Offset,PR[24:Rotate_Offset] ;
 531:L P[441]  R[157] mm/sec CNT100 Offset,PR[24:Rotate_Offset] ;
 532:L P[442]  R[157] mm/sec CNT100 Offset,PR[24:Rotate_Offset] ;
 533:L P[443]  R[157] mm/sec CNT100 Offset,PR[24:Rotate_Offset] ;
 534:L P[444]  R[157] mm/sec CNT100 Offset,PR[24:Rotate_Offset] ;
 535: !Pass12 ;
 536: LBL[112:Pass12] ;
 537:L P[445]  R[157] mm/sec FINE Offset,PR[78:Offst_apprch]  ;
 538: WAIT   0.20(sec) ;
 539:L P[445]  R[157] mm/sec CNT100 TA    0.00sec,CALL RUN_LASER_START Offset,PR[25:Start_Offset] ;
 541:L P[446]  R[157] mm/sec CNT100 Offset,PR[24:Rotate_Offset] ;
 542:L P[447]  R[157] mm/sec CNT100 Offset,PR[24:Rotate_Offset] ;
 543:L P[448]  R[157] mm/sec CNT100 Offset,PR[24:Rotate_Offset] ;
 544:L P[449]  R[157] mm/sec CNT100 Offset,PR[24:Rotate_Offset] ;
 545:L P[450]  R[157] mm/sec CNT100 Offset,PR[24:Rotate_Offset] ;
 546:L P[451]  R[157] mm/sec CNT100 Offset,PR[24:Rotate_Offset] ;
 547:L P[452]  R[157] mm/sec CNT100 TA    0.00sec,CALL RUN_LASER_STOP Offset,PR[26:Stop_Offset] ;
 549:L P[452]  R[157] mm/sec FINE Offset,PR[76:Offst_dprt] ;
 550:L P[453]  R[157] mm/sec CNT100 Offset,PR[24:Rotate_Offset] ;
 551:L P[454]  R[157] mm/sec CNT100 Offset,PR[24:Rotate_Offset] ;
 552:L P[455]  R[157] mm/sec CNT100 Offset,PR[24:Rotate_Offset] ;
 553:L P[456]  R[157] mm/sec CNT100 Offset,PR[24:Rotate_Offset] ;
 554:L P[457]  R[157] mm/sec CNT100 Offset,PR[24:Rotate_Offset] ;
 555:L P[458]  R[157] mm/sec CNT100 Offset,PR[24:Rotate_Offset] ;
 556: !Pass13 ;
 557: LBL[113:Pass13] ;
 558:L P[459]  R[157] mm/sec FINE Offset,PR[78:Offst_apprch]  ;
 559: WAIT   0.20(sec) ;
 560:L P[459]  R[157] mm/sec CNT100 TA    0.00sec,CALL RUN_LASER_START Offset,PR[25:Start_Offset] ;
 562:L P[460]  R[157] mm/sec CNT100 Offset,PR[24:Rotate_Offset] ;
 563:L P[461]  R[157] mm/sec CNT100 Offset,PR[24:Rotate_Offset] ;
 564:L P[462]  R[157] mm/sec CNT100 Offset,PR[24:Rotate_Offset] ;
 565:L P[463]  R[157] mm/sec CNT100 Offset,PR[24:Rotate_Offset] ;
 566:L P[464]  R[157] mm/sec CNT100 Offset,PR[24:Rotate_Offset] ;
 567:L P[465]  R[157] mm/sec CNT100 Offset,PR[24:Rotate_Offset] ;
 568:L P[466]  R[157] mm/sec CNT100 Offset,PR[24:Rotate_Offset] ;
 569:L P[467]  R[157] mm/sec CNT100 Offset,PR[24:Rotate_Offset] ;
 570:L P[468]  R[157] mm/sec CNT100 Offset,PR[24:Rotate_Offset] ;
 571:L P[469]  R[157] mm/sec CNT100 Offset,PR[24:Rotate_Offset] ;
 572:L P[470]  R[157] mm/sec CNT100 Offset,PR[24:Rotate_Offset] ;
 573:L P[471]  R[157] mm/sec CNT100 Offset,PR[24:Rotate_Offset] ;
 574:L P[472]  R[157] mm/sec CNT100 Offset,PR[24:Rotate_Offset] ;
 575:L P[473]  R[157] mm/sec CNT100 TA    0.00sec,CALL RUN_LASER_STOP Offset,PR[26:Stop_Offset] ;
 577:L P[473]  R[157] mm/sec FINE Offset,PR[76:Offst_dprt] ;
 578:L P[474]  R[157] mm/sec CNT100 Offset,PR[24:Rotate_Offset] ;
 579:L P[475]  R[157] mm/sec CNT100 Offset,PR[24:Rotate_Offset] ;
 580:L P[476]  R[157] mm/sec CNT100 Offset,PR[24:Rotate_Offset] ;
 581:L P[477]  R[157] mm/sec CNT100 Offset,PR[24:Rotate_Offset] ;
 582:L P[478]  R[157] mm/sec CNT100 Offset,PR[24:Rotate_Offset] ;
 583:L P[479]  R[157] mm/sec CNT100 Offset,PR[24:Rotate_Offset] ;
 584: !Pass14 ;
 585: LBL[114:Pass14] ;
 586:L P[480]  R[157] mm/sec FINE Offset,PR[78:Offst_apprch]  ;
 587: WAIT   0.20(sec) ;
 588:L P[480]  R[157] mm/sec CNT100 TA    0.00sec,CALL RUN_LASER_START Offset,PR[25:Start_Offset] ;
 590:L P[481]  R[157] mm/sec CNT100 Offset,PR[24:Rotate_Offset] ;
 591:L P[482]  R[157] mm/sec CNT100 Offset,PR[24:Rotate_Offset] ;
 592:L P[483]  R[157] mm/sec CNT100 Offset,PR[24:Rotate_Offset] ;
 593:L P[484]  R[157] mm/sec CNT100 Offset,PR[24:Rotate_Offset] ;
 594:L P[485]  R[157] mm/sec CNT100 Offset,PR[24:Rotate_Offset] ;
 595:L P[486]  R[157] mm/sec CNT100 TA    0.00sec,CALL RUN_LASER_STOP Offset,PR[26:Stop_Offset] ;
 597:L P[486]  R[157] mm/sec FINE Offset,PR[76:Offst_dprt] ;
 598:L P[487]  R[157] mm/sec CNT100 Offset,PR[24:Rotate_Offset] ;
 599:L P[488]  R[157] mm/sec CNT100 Offset,PR[24:Rotate_Offset] ;
 600:L P[489]  R[157] mm/sec CNT100 Offset,PR[24:Rotate_Offset] ;
 601:L P[490]  R[157] mm/sec CNT100 Offset,PR[24:Rotate_Offset] ;
 602:L P[491]  R[157] mm/sec CNT100 Offset,PR[24:Rotate_Offset] ;
 603:L P[492]  R[157] mm/sec CNT100 Offset,PR[24:Rotate_Offset] ;
 604: !Pass15 ;
 605: LBL[115:Pass15] ;
 606:L P[493]  R[157] mm/sec FINE Offset,PR[78:Offst_apprch]  ;
 607: WAIT   0.20(sec) ;
 608:L P[493]  R[157] mm/sec CNT100 TA    0.00sec,CALL RUN_LASER_START Offset,PR[25:Start_Offset] ;
 610:L P[494]  R[157] mm/sec CNT100 Offset,PR[24:Rotate_Offset] ;
 611:L P[495]  R[157] mm/sec CNT100 Offset,PR[24:Rotate_Offset] ;
 612:L P[496]  R[157] mm/sec CNT100 Offset,PR[24:Rotate_Offset] ;
 613:L P[497]  R[157] mm/sec CNT100 Offset,PR[24:Rotate_Offset] ;
 614:L P[498]  R[157] mm/sec CNT100 Offset,PR[24:Rotate_Offset] ;
 615:L P[499]  R[157] mm/sec CNT100 Offset,PR[24:Rotate_Offset] ;
 616:L P[500]  R[157] mm/sec CNT100 Offset,PR[24:Rotate_Offset] ;
 617:L P[501]  R[157] mm/sec CNT100 Offset,PR[24:Rotate_Offset] ;
 618:L P[502]  R[157] mm/sec CNT100 Offset,PR[24:Rotate_Offset] ;
 619:L P[503]  R[157] mm/sec CNT100 Offset,PR[24:Rotate_Offset] ;
 620:L P[504]  R[157] mm/sec CNT100 Offset,PR[24:Rotate_Offset] ;
 621:L P[505]  R[157] mm/sec CNT100 Offset,PR[24:Rotate_Offset] ;
 622:L P[506]  R[157] mm/sec CNT100 Offset,PR[24:Rotate_Offset] ;
 623:L P[507]  R[157] mm/sec CNT100 Offset,PR[24:Rotate_Offset] ;
 624:L P[508]  R[157] mm/sec CNT100 Offset,PR[24:Rotate_Offset] ;
 625:L P[509]  R[157] mm/sec CNT100 TA    0.00sec,CALL RUN_LASER_STOP Offset,PR[26:Stop_Offset] ;
 627:L P[509]  R[157] mm/sec FINE Offset,PR[76:Offst_dprt] ;
 628:L P[510]  R[157] mm/sec CNT100 Offset,PR[24:Rotate_Offset] ;
 629:L P[511]  R[157] mm/sec CNT100 Offset,PR[24:Rotate_Offset] ;
 630:L P[512]  R[157] mm/sec CNT100 Offset,PR[24:Rotate_Offset] ;
 631:L P[513]  R[157] mm/sec CNT100 Offset,PR[24:Rotate_Offset] ;
 632:L P[514]  R[157] mm/sec CNT100 Offset,PR[24:Rotate_Offset] ;
 633:L P[515]  R[157] mm/sec CNT100 Offset,PR[24:Rotate_Offset] ;
 634: !Pass16 ;
 635: LBL[116:Pass16] ;
 636:L P[516]  R[157] mm/sec FINE Offset,PR[78:Offst_apprch]  ;
 637: WAIT   0.20(sec) ;
 638:L P[516]  R[157] mm/sec CNT100 TA    0.00sec,CALL RUN_LASER_START Offset,PR[25:Start_Offset] ;
 640:L P[517]  R[157] mm/sec CNT100 Offset,PR[24:Rotate_Offset] ;
 641:L P[518]  R[157] mm/sec CNT100 Offset,PR[24:Rotate_Offset] ;
 642:L P[519]  R[157] mm/sec CNT100 Offset,PR[24:Rotate_Offset] ;
 643:L P[520]  R[157] mm/sec CNT100 Offset,PR[24:Rotate_Offset] ;
 644:L P[521]  R[157] mm/sec CNT100 Offset,PR[24:Rotate_Offset] ;
 645:L P[522]  R[157] mm/sec CNT100 Offset,PR[24:Rotate_Offset] ;
 646:L P[523]  R[157] mm/sec CNT100 Offset,PR[24:Rotate_Offset] ;
 647:L P[524]  R[157] mm/sec CNT100 TA    0.00sec,CALL RUN_LASER_STOP Offset,PR[26:Stop_Offset] ;
 649:L P[524]  R[157] mm/sec FINE Offset,PR[76:Offst_dprt] ;
 650:L P[525]  R[157] mm/sec CNT100 Offset,PR[24:Rotate_Offset] ;
 651:L P[526]  R[157] mm/sec CNT100 Offset,PR[24:Rotate_Offset] ;
 652:L P[527]  R[157] mm/sec CNT100 Offset,PR[24:Rotate_Offset] ;
 653:L P[528]  R[157] mm/sec CNT100 Offset,PR[24:Rotate_Offset] ;
 654:L P[529]  R[157] mm/sec CNT100 Offset,PR[24:Rotate_Offset] ;
 655:L P[530]  R[157] mm/sec CNT100 Offset,PR[24:Rotate_Offset] ;
 656: !Pass17 ;
 657: LBL[117:Pass17] ;
 658:L P[531]  R[157] mm/sec FINE Offset,PR[78:Offst_apprch]  ;
 659: WAIT   0.20(sec) ;
 660:L P[531]  R[157] mm/sec CNT100 TA    0.00sec,CALL RUN_LASER_START Offset,PR[25:Start_Offset] ;
 662:L P[532]  R[157] mm/sec CNT100 Offset,PR[24:Rotate_Offset] ;
 663:L P[533]  R[157] mm/sec CNT100 Offset,PR[24:Rotate_Offset] ;
 664:L P[534]  R[157] mm/sec CNT100 Offset,PR[24:Rotate_Offset] ;
 665:L P[535]  R[157] mm/sec CNT100 Offset,PR[24:Rotate_Offset] ;
 666:L P[536]  R[157] mm/sec CNT100 Offset,PR[24:Rotate_Offset] ;
 667:L P[537]  R[157] mm/sec CNT100 Offset,PR[24:Rotate_Offset] ;
 668:L P[538]  R[157] mm/sec CNT100 Offset,PR[24:Rotate_Offset] ;
 669:L P[539]  R[157] mm/sec CNT100 Offset,PR[24:Rotate_Offset] ;
 670:L P[540]  R[157] mm/sec CNT100 TA    0.00sec,CALL RUN_LASER_STOP Offset,PR[26:Stop_Offset] ;
 672:L P[540]  R[157] mm/sec FINE Offset,PR[76:Offst_dprt] ;
 673:L P[541]  R[157] mm/sec CNT100 Offset,PR[24:Rotate_Offset] ;
 674:L P[542]  R[157] mm/sec CNT100 Offset,PR[24:Rotate_Offset] ;
 675:L P[543]  R[157] mm/sec CNT100 Offset,PR[24:Rotate_Offset] ;
 676:L P[544]  R[157] mm/sec CNT100 Offset,PR[24:Rotate_Offset] ;
 677:L P[545]  R[157] mm/sec CNT100 Offset,PR[24:Rotate_Offset] ;
 678:L P[546]  R[157] mm/sec CNT100 Offset,PR[24:Rotate_Offset] ;
 679: !Pass18 ;
 680: LBL[118:Pass18] ;
 681:L P[547]  R[157] mm/sec FINE Offset,PR[78:Offst_apprch]  ;
 682: WAIT   0.20(sec) ;
 683:L P[547]  R[157] mm/sec CNT100 TA    0.00sec,CALL RUN_LASER_START Offset,PR[25:Start_Offset] ;
 685:L P[548]  R[157] mm/sec CNT100 Offset,PR[24:Rotate_Offset] ;
 686:L P[549]  R[157] mm/sec CNT100 Offset,PR[24:Rotate_Offset] ;
 687:L P[550]  R[157] mm/sec CNT100 Offset,PR[24:Rotate_Offset] ;
 688:L P[551]  R[157] mm/sec CNT100 Offset,PR[24:Rotate_Offset] ;
 689:L P[552]  R[157] mm/sec CNT100 Offset,PR[24:Rotate_Offset] ;
 690:L P[553]  R[157] mm/sec CNT100 Offset,PR[24:Rotate_Offset] ;
 691:L P[554]  R[157] mm/sec CNT100 Offset,PR[24:Rotate_Offset] ;
 692:L P[555]  R[157] mm/sec CNT100 Offset,PR[24:Rotate_Offset] ;
 693:L P[556]  R[157] mm/sec CNT100 Offset,PR[24:Rotate_Offset] ;
 694:L P[557]  R[157] mm/sec CNT100 Offset,PR[24:Rotate_Offset] ;
 695:L P[558]  R[157] mm/sec CNT100 Offset,PR[24:Rotate_Offset] ;
 696:L P[559]  R[157] mm/sec CNT100 Offset,PR[24:Rotate_Offset] ;
 697:L P[560]  R[157] mm/sec CNT100 Offset,PR[24:Rotate_Offset] ;
 698:L P[561]  R[157] mm/sec CNT100 Offset,PR[24:Rotate_Offset] ;
 699:L P[562]  R[157] mm/sec CNT100 TA    0.00sec,CALL RUN_LASER_STOP Offset,PR[26:Stop_Offset] ;
 701:L P[562]  R[157] mm/sec FINE Offset,PR[76:Offst_dprt] ;
 702:L P[563]  R[157] mm/sec CNT100 Offset,PR[24:Rotate_Offset] ;
 703:L P[564]  R[157] mm/sec CNT100 Offset,PR[24:Rotate_Offset] ;
 704:L P[565]  R[157] mm/sec CNT100 Offset,PR[24:Rotate_Offset] ;
 705:L P[566]  R[157] mm/sec CNT100 Offset,PR[24:Rotate_Offset] ;
 706:L P[567]  R[157] mm/sec CNT100 Offset,PR[24:Rotate_Offset] ;
 707:L P[568]  R[157] mm/sec CNT100 Offset,PR[24:Rotate_Offset] ;
 708: !Pass19 ;
 709: LBL[119:Pass19] ;
 710:L P[569]  R[157] mm/sec FINE Offset,PR[78:Offst_apprch]  ;
 711: WAIT   0.20(sec) ;
 712:L P[569]  R[157] mm/sec CNT100 TA    0.00sec,CALL RUN_LASER_START Offset,PR[25:Start_Offset] ;
 714:L P[570]  R[157] mm/sec CNT100 Offset,PR[24:Rotate_Offset] ;
 715:L P[571]  R[157] mm/sec CNT100 Offset,PR[24:Rotate_Offset] ;
 716:L P[572]  R[157] mm/sec CNT100 Offset,PR[24:Rotate_Offset] ;
 717:L P[573]  R[157] mm/sec CNT100 Offset,PR[24:Rotate_Offset] ;
 718:L P[574]  R[157] mm/sec CNT100 Offset,PR[24:Rotate_Offset] ;
 719:L P[575]  R[157] mm/sec CNT100 TA    0.00sec,CALL RUN_LASER_STOP Offset,PR[26:Stop_Offset] ;
 721:L P[575]  R[157] mm/sec FINE Offset,PR[76:Offst_dprt] ;
 722:L P[576]  R[157] mm/sec CNT100 Offset,PR[24:Rotate_Offset] ;
 723:L P[577]  R[157] mm/sec CNT100 Offset,PR[24:Rotate_Offset] ;
 724:L P[578]  R[157] mm/sec CNT100 Offset,PR[24:Rotate_Offset] ;
 725:L P[579]  R[157] mm/sec CNT100 Offset,PR[24:Rotate_Offset] ;
 726:L P[580]  R[157] mm/sec CNT100 Offset,PR[24:Rotate_Offset] ;
 727:L P[581]  R[157] mm/sec CNT100 Offset,PR[24:Rotate_Offset] ;
 728: !Pass20 ;
 729: LBL[120:Pass20] ;
 730:L P[582]  R[157] mm/sec FINE Offset,PR[78:Offst_apprch]  ;
 731: WAIT   0.20(sec) ;
 732:L P[582]  R[157] mm/sec CNT100 TA    0.00sec,CALL RUN_LASER_START Offset,PR[25:Start_Offset] ;
 734:L P[583]  R[157] mm/sec CNT100 Offset,PR[24:Rotate_Offset] ;
 735:L P[584]  R[157] mm/sec CNT100 Offset,PR[24:Rotate_Offset] ;
 736:L P[585]  R[157] mm/sec CNT100 Offset,PR[24:Rotate_Offset] ;
 737:L P[586]  R[157] mm/sec CNT100 Offset,PR[24:Rotate_Offset] ;
 738:L P[587]  R[157] mm/sec CNT100 Offset,PR[24:Rotate_Offset] ;
 739:L P[588]  R[157] mm/sec CNT100 Offset,PR[24:Rotate_Offset] ;
 740:L P[589]  R[157] mm/sec CNT100 Offset,PR[24:Rotate_Offset] ;
 741:L P[590]  R[157] mm/sec CNT100 Offset,PR[24:Rotate_Offset] ;
 742:L P[591]  R[157] mm/sec CNT100 Offset,PR[24:Rotate_Offset] ;
 743:L P[592]  R[157] mm/sec CNT100 Offset,PR[24:Rotate_Offset] ;
 744:L P[593]  R[157] mm/sec CNT100 Offset,PR[24:Rotate_Offset] ;
 745:L P[594]  R[157] mm/sec CNT100 Offset,PR[24:Rotate_Offset] ;
 746:L P[595]  R[157] mm/sec CNT100 Offset,PR[24:Rotate_Offset] ;
 747:L P[596]  R[157] mm/sec CNT100 TA    0.00sec,CALL RUN_LASER_STOP Offset,PR[26:Stop_Offset] ;
 749:L P[596]  R[157] mm/sec FINE Offset,PR[76:Offst_dprt] ;
 750:L P[597]  R[157] mm/sec CNT100 Offset,PR[24:Rotate_Offset] ;
 751:L P[598]  R[157] mm/sec CNT100 Offset,PR[24:Rotate_Offset] ;
 752:L P[599]  R[157] mm/sec CNT100 Offset,PR[24:Rotate_Offset] ;
 753:L P[600]  R[157] mm/sec CNT100 Offset,PR[24:Rotate_Offset] ;
 754:L P[601]  R[157] mm/sec CNT100 Offset,PR[24:Rotate_Offset] ;
 755:L P[602]  R[157] mm/sec CNT100 Offset,PR[24:Rotate_Offset] ;
 756: !Pass21 ;
 757: LBL[121:Pass21] ;
 758:L P[603]  R[157] mm/sec FINE Offset,PR[78:Offst_apprch]  ;
 759: WAIT   0.20(sec) ;
 760:L P[603]  R[157] mm/sec CNT100 TA    0.00sec,CALL RUN_LASER_START Offset,PR[25:Start_Offset] ;
 762:L P[604]  R[157] mm/sec CNT100 Offset,PR[24:Rotate_Offset] ;
 763:L P[605]  R[157] mm/sec CNT100 Offset,PR[24:Rotate_Offset] ;
 764:L P[606]  R[157] mm/sec CNT100 Offset,PR[24:Rotate_Offset] ;
 765:L P[607]  R[157] mm/sec CNT100 Offset,PR[24:Rotate_Offset] ;
 766:L P[608]  R[157] mm/sec CNT100 Offset,PR[24:Rotate_Offset] ;
 767:L P[609]  R[157] mm/sec CNT100 Offset,PR[24:Rotate_Offset] ;
 768:L P[610]  R[157] mm/sec CNT100 TA    0.00sec,CALL RUN_LASER_STOP Offset,PR[26:Stop_Offset] ;
 770:L P[610]  R[157] mm/sec FINE Offset,PR[76:Offst_dprt] ;
 771:L P[611]  R[157] mm/sec CNT100 Offset,PR[24:Rotate_Offset] ;
 772:L P[612]  R[157] mm/sec CNT100 Offset,PR[24:Rotate_Offset] ;
 773:L P[613]  R[157] mm/sec CNT100 Offset,PR[24:Rotate_Offset] ;
 774:L P[614]  R[157] mm/sec CNT100 Offset,PR[24:Rotate_Offset] ;
 775:L P[615]  R[157] mm/sec CNT100 Offset,PR[24:Rotate_Offset] ;
 776:L P[616]  R[157] mm/sec CNT100 Offset,PR[24:Rotate_Offset] ;
 777: !Pass22 ;
 778: LBL[122:Pass22] ;
 779:L P[617]  R[157] mm/sec FINE Offset,PR[78:Offst_apprch]  ;
 780: WAIT   0.20(sec) ;
 781:L P[617]  R[157] mm/sec CNT100 TA    0.00sec,CALL RUN_LASER_START Offset,PR[25:Start_Offset] ;
 783:L P[618]  R[157] mm/sec CNT100 Offset,PR[24:Rotate_Offset] ;
 784:L P[619]  R[157] mm/sec CNT100 Offset,PR[24:Rotate_Offset] ;
 785:L P[620]  R[157] mm/sec CNT100 Offset,PR[24:Rotate_Offset] ;
 786:L P[621]  R[157] mm/sec CNT100 Offset,PR[24:Rotate_Offset] ;
 787:L P[622]  R[157] mm/sec CNT100 Offset,PR[24:Rotate_Offset] ;
 788:L P[623]  R[157] mm/sec CNT100 TA    0.00sec,CALL RUN_LASER_STOP Offset,PR[26:Stop_Offset] ;
 790:L P[623]  R[157] mm/sec FINE Offset,PR[76:Offst_dprt] ;
 791:L P[624]  R[157] mm/sec CNT100 Offset,PR[24:Rotate_Offset] ;
 792:L P[625]  R[157] mm/sec CNT100 Offset,PR[24:Rotate_Offset] ;
 793:L P[626]  R[157] mm/sec CNT100 Offset,PR[24:Rotate_Offset] ;
 794:L P[627]  R[157] mm/sec CNT100 Offset,PR[24:Rotate_Offset] ;
 795:L P[628]  R[157] mm/sec CNT100 Offset,PR[24:Rotate_Offset] ;
 796:L P[629]  R[157] mm/sec CNT100 Offset,PR[24:Rotate_Offset] ;
 797: !Pass23 ;
 798: LBL[123:Pass23] ;
 799:L P[630]  R[157] mm/sec FINE Offset,PR[78:Offst_apprch]  ;
 800: WAIT   0.20(sec) ;
 801:L P[630]  R[157] mm/sec CNT100 TA    0.00sec,CALL RUN_LASER_START Offset,PR[25:Start_Offset] ;
 803:L P[631]  R[157] mm/sec CNT100 Offset,PR[24:Rotate_Offset] ;
 804:L P[632]  R[157] mm/sec CNT100 Offset,PR[24:Rotate_Offset] ;
 805:L P[633]  R[157] mm/sec CNT100 Offset,PR[24:Rotate_Offset] ;
 806:L P[634]  R[157] mm/sec CNT100 Offset,PR[24:Rotate_Offset] ;
 807:L P[635]  R[157] mm/sec CNT100 Offset,PR[24:Rotate_Offset] ;
 808:L P[636]  R[157] mm/sec CNT100 Offset,PR[24:Rotate_Offset] ;
 809:L P[637]  R[157] mm/sec CNT100 Offset,PR[24:Rotate_Offset] ;
 810:L P[638]  R[157] mm/sec CNT100 Offset,PR[24:Rotate_Offset] ;
 811:L P[639]  R[157] mm/sec CNT100 Offset,PR[24:Rotate_Offset] ;
 812:L P[640]  R[157] mm/sec CNT100 Offset,PR[24:Rotate_Offset] ;
 813:L P[641]  R[157] mm/sec CNT100 Offset,PR[24:Rotate_Offset] ;
 814:L P[642]  R[157] mm/sec CNT100 TA    0.00sec,CALL RUN_LASER_STOP Offset,PR[26:Stop_Offset] ;
 816:L P[642]  R[157] mm/sec FINE Offset,PR[76:Offst_dprt] ;
 817:L P[643]  R[157] mm/sec CNT100 Offset,PR[24:Rotate_Offset] ;
 818:L P[644]  R[157] mm/sec CNT100 Offset,PR[24:Rotate_Offset] ;
 819:L P[645]  R[157] mm/sec CNT100 Offset,PR[24:Rotate_Offset] ;
 820:L P[646]  R[157] mm/sec CNT100 Offset,PR[24:Rotate_Offset] ;
 821:L P[647]  R[157] mm/sec CNT100 Offset,PR[24:Rotate_Offset] ;
 822:L P[648]  R[157] mm/sec CNT100 Offset,PR[24:Rotate_Offset] ;
 823: !Pass24 ;
 824: LBL[124:Pass24] ;
 825:L P[649]  R[157] mm/sec FINE Offset,PR[78:Offst_apprch]  ;
 826: WAIT   0.20(sec) ;
 827:L P[649]  R[157] mm/sec CNT100 TA    0.00sec,CALL RUN_LASER_START Offset,PR[25:Start_Offset] ;
 829:L P[650]  R[157] mm/sec CNT100 Offset,PR[24:Rotate_Offset] ;
 830:L P[651]  R[157] mm/sec CNT100 Offset,PR[24:Rotate_Offset] ;
 831:L P[652]  R[157] mm/sec CNT100 Offset,PR[24:Rotate_Offset] ;
 832:L P[653]  R[157] mm/sec CNT100 Offset,PR[24:Rotate_Offset] ;
 833:L P[654]  R[157] mm/sec CNT100 Offset,PR[24:Rotate_Offset] ;
 834:L P[655]  R[157] mm/sec CNT100 TA    0.00sec,CALL RUN_LASER_STOP Offset,PR[26:Stop_Offset] ;
 836:L P[655]  R[157] mm/sec FINE Offset,PR[76:Offst_dprt] ;
 837:L P[656]  R[157] mm/sec CNT100 Offset,PR[24:Rotate_Offset] ;
 838:L P[657]  R[157] mm/sec CNT100 Offset,PR[24:Rotate_Offset] ;
 839:L P[658]  R[157] mm/sec CNT100 Offset,PR[24:Rotate_Offset] ;
 840:L P[659]  R[157] mm/sec CNT100 Offset,PR[24:Rotate_Offset] ;
 841:L P[660]  R[157] mm/sec CNT100 Offset,PR[24:Rotate_Offset] ;
 842:L P[661]  R[157] mm/sec CNT100 Offset,PR[24:Rotate_Offset] ;
 843: !Pass25 ;
 844: LBL[125:Pass25] ;
 845:L P[662]  R[157] mm/sec FINE Offset,PR[78:Offst_apprch]  ;
 846: WAIT   0.20(sec) ;
 847:L P[662]  R[157] mm/sec CNT100 TA    0.00sec,CALL RUN_LASER_START Offset,PR[25:Start_Offset] ;
 849:L P[663]  R[157] mm/sec CNT100 Offset,PR[24:Rotate_Offset] ;
 850:L P[664]  R[157] mm/sec CNT100 Offset,PR[24:Rotate_Offset] ;
 851:L P[665]  R[157] mm/sec CNT100 Offset,PR[24:Rotate_Offset] ;
 852:L P[666]  R[157] mm/sec CNT100 Offset,PR[24:Rotate_Offset] ;
 853:L P[667]  R[157] mm/sec CNT100 Offset,PR[24:Rotate_Offset] ;
 854:L P[668]  R[157] mm/sec CNT100 Offset,PR[24:Rotate_Offset] ;
 855:L P[669]  R[157] mm/sec CNT100 Offset,PR[24:Rotate_Offset] ;
 856:L P[670]  R[157] mm/sec CNT100 Offset,PR[24:Rotate_Offset] ;
 857:L P[671]  R[157] mm/sec CNT100 Offset,PR[24:Rotate_Offset] ;
 858:L P[672]  R[157] mm/sec CNT100 Offset,PR[24:Rotate_Offset] ;
 859:L P[673]  R[157] mm/sec CNT100 Offset,PR[24:Rotate_Offset] ;
 860:L P[674]  R[157] mm/sec CNT100 Offset,PR[24:Rotate_Offset] ;
 861:L P[675]  R[157] mm/sec CNT100 Offset,PR[24:Rotate_Offset] ;
 862:L P[676]  R[157] mm/sec CNT100 Offset,PR[24:Rotate_Offset] ;
 863:L P[677]  R[157] mm/sec CNT100 Offset,PR[24:Rotate_Offset] ;
 864:L P[678]  R[157] mm/sec CNT100 TA    0.00sec,CALL RUN_LASER_STOP Offset,PR[26:Stop_Offset] ;
 866:L P[678]  R[157] mm/sec FINE Offset,PR[76:Offst_dprt] ;
 867:L P[679]  R[157] mm/sec CNT100 Offset,PR[24:Rotate_Offset] ;
 868:L P[680]  R[157] mm/sec CNT100 Offset,PR[24:Rotate_Offset] ;
 869:L P[681]  R[157] mm/sec CNT100 Offset,PR[24:Rotate_Offset] ;
 870:L P[682]  R[157] mm/sec CNT100 Offset,PR[24:Rotate_Offset] ;
 871:L P[683]  R[157] mm/sec CNT100 Offset,PR[24:Rotate_Offset] ;
 872:L P[684]  R[157] mm/sec CNT100 Offset,PR[24:Rotate_Offset] ;
 873: !Pass26 ;
 874: LBL[126:Pass26] ;
 875:L P[685]  R[157] mm/sec FINE Offset,PR[78:Offst_apprch]  ;
 876: WAIT   0.20(sec) ;
 877:L P[685]  R[157] mm/sec CNT100 TA    0.00sec,CALL RUN_LASER_START Offset,PR[25:Start_Offset] ;
 879:L P[686]  R[157] mm/sec CNT100 Offset,PR[24:Rotate_Offset] ;
 880:L P[687]  R[157] mm/sec CNT100 Offset,PR[24:Rotate_Offset] ;
 881:L P[688]  R[157] mm/sec CNT100 Offset,PR[24:Rotate_Offset] ;
 882:L P[689]  R[157] mm/sec CNT100 Offset,PR[24:Rotate_Offset] ;
 883:L P[690]  R[157] mm/sec CNT100 Offset,PR[24:Rotate_Offset] ;
 884:L P[691]  R[157] mm/sec CNT100 Offset,PR[24:Rotate_Offset] ;
 885:L P[692]  R[157] mm/sec CNT100 Offset,PR[24:Rotate_Offset] ;
 886:L P[693]  R[157] mm/sec CNT100 Offset,PR[24:Rotate_Offset] ;
 887:L P[694]  R[157] mm/sec CNT100 TA    0.00sec,CALL RUN_LASER_STOP Offset,PR[26:Stop_Offset] ;
 889:L P[694]  R[157] mm/sec FINE Offset,PR[76:Offst_dprt] ;
 890:L P[695]  R[157] mm/sec CNT100 Offset,PR[24:Rotate_Offset] ;
 891:L P[696]  R[157] mm/sec CNT100 Offset,PR[24:Rotate_Offset] ;
 892:L P[697]  R[157] mm/sec CNT100 Offset,PR[24:Rotate_Offset] ;
 893:L P[698]  R[157] mm/sec CNT100 Offset,PR[24:Rotate_Offset] ;
 894:L P[699]  R[157] mm/sec CNT100 Offset,PR[24:Rotate_Offset] ;
 895:L P[700]  R[157] mm/sec CNT100 Offset,PR[24:Rotate_Offset] ;
 896: !Pass27 ;
 897: LBL[127:Pass27] ;
 898:L P[701]  R[157] mm/sec FINE Offset,PR[78:Offst_apprch]  ;
 899: WAIT   0.20(sec) ;
 900:L P[701]  R[157] mm/sec CNT100 TA    0.00sec,CALL RUN_LASER_START Offset,PR[25:Start_Offset] ;
 902:L P[702]  R[157] mm/sec CNT100 Offset,PR[24:Rotate_Offset] ;
 903:L P[703]  R[157] mm/sec CNT100 Offset,PR[24:Rotate_Offset] ;
 904:L P[704]  R[157] mm/sec CNT100 Offset,PR[24:Rotate_Offset] ;
 905:L P[705]  R[157] mm/sec CNT100 Offset,PR[24:Rotate_Offset] ;
 906:L P[706]  R[157] mm/sec CNT100 Offset,PR[24:Rotate_Offset] ;
 907:L P[707]  R[157] mm/sec CNT100 Offset,PR[24:Rotate_Offset] ;
 908:L P[708]  R[157] mm/sec CNT100 Offset,PR[24:Rotate_Offset] ;
 909:L P[709]  R[157] mm/sec CNT100 Offset,PR[24:Rotate_Offset] ;
 910:L P[710]  R[157] mm/sec CNT100 Offset,PR[24:Rotate_Offset] ;
 911:L P[711]  R[157] mm/sec CNT100 TA    0.00sec,CALL RUN_LASER_STOP Offset,PR[26:Stop_Offset] ;
 913:L P[711]  R[157] mm/sec FINE Offset,PR[76:Offst_dprt] ;
 914:L P[712]  R[157] mm/sec CNT100 Offset,PR[24:Rotate_Offset] ;
 915:L P[713]  R[157] mm/sec CNT100 Offset,PR[24:Rotate_Offset] ;
 916:L P[714]  R[157] mm/sec CNT100 Offset,PR[24:Rotate_Offset] ;
 917:L P[715]  R[157] mm/sec CNT100 Offset,PR[24:Rotate_Offset] ;
 918:L P[716]  R[157] mm/sec CNT100 Offset,PR[24:Rotate_Offset] ;
 919:L P[717]  R[157] mm/sec CNT100 Offset,PR[24:Rotate_Offset] ;
 920: !Pass28 ;
 921: LBL[128:Pass28] ;
 922:L P[718]  R[157] mm/sec FINE Offset,PR[78:Offst_apprch]  ;
 923: WAIT   0.20(sec) ;
 924:L P[718]  R[157] mm/sec CNT100 TA    0.00sec,CALL RUN_LASER_START Offset,PR[25:Start_Offset] ;
 926:L P[719]  R[157] mm/sec CNT100 Offset,PR[24:Rotate_Offset] ;
 927:L P[720]  R[157] mm/sec CNT100 Offset,PR[24:Rotate_Offset] ;
 928:L P[721]  R[157] mm/sec CNT100 Offset,PR[24:Rotate_Offset] ;
 929:L P[722]  R[157] mm/sec CNT100 Offset,PR[24:Rotate_Offset] ;
 930:L P[723]  R[157] mm/sec CNT100 Offset,PR[24:Rotate_Offset] ;
 931:L P[724]  R[157] mm/sec CNT100 Offset,PR[24:Rotate_Offset] ;
 932:L P[725]  R[157] mm/sec CNT100 Offset,PR[24:Rotate_Offset] ;
 933:L P[726]  R[157] mm/sec CNT100 Offset,PR[24:Rotate_Offset] ;
 934:L P[727]  R[157] mm/sec CNT100 Offset,PR[24:Rotate_Offset] ;
 935:L P[728]  R[157] mm/sec CNT100 Offset,PR[24:Rotate_Offset] ;
 936:L P[729]  R[157] mm/sec CNT100 Offset,PR[24:Rotate_Offset] ;
 937:L P[730]  R[157] mm/sec CNT100 Offset,PR[24:Rotate_Offset] ;
 938:L P[731]  R[157] mm/sec CNT100 Offset,PR[24:Rotate_Offset] ;
 939:L P[732]  R[157] mm/sec CNT100 Offset,PR[24:Rotate_Offset] ;
 940:L P[733]  R[157] mm/sec CNT100 Offset,PR[24:Rotate_Offset] ;
 941:L P[734]  R[157] mm/sec CNT100 TA    0.00sec,CALL RUN_LASER_STOP Offset,PR[26:Stop_Offset] ;
 943:L P[734]  R[157] mm/sec FINE Offset,PR[76:Offst_dprt] ;
 944:L P[735]  R[157] mm/sec CNT100 Offset,PR[24:Rotate_Offset] ;
 945:L P[736]  R[157] mm/sec CNT100 Offset,PR[24:Rotate_Offset] ;
 946:L P[737]  R[157] mm/sec CNT100 Offset,PR[24:Rotate_Offset] ;
 947:L P[738]  R[157] mm/sec CNT100 Offset,PR[24:Rotate_Offset] ;
 948:L P[739]  R[157] mm/sec CNT100 Offset,PR[24:Rotate_Offset] ;
 949:L P[740]  R[157] mm/sec CNT100 Offset,PR[24:Rotate_Offset] ;
 950: !Pass29 ;
 951: LBL[129:Pass29] ;
 952:L P[741]  R[157] mm/sec FINE Offset,PR[78:Offst_apprch]  ;
 953: WAIT   0.20(sec) ;
 954:L P[741]  R[157] mm/sec CNT100 TA    0.00sec,CALL RUN_LASER_START Offset,PR[25:Start_Offset] ;
 956:L P[742]  R[157] mm/sec CNT100 Offset,PR[24:Rotate_Offset] ;
 957:L P[743]  R[157] mm/sec CNT100 Offset,PR[24:Rotate_Offset] ;
 958:L P[744]  R[157] mm/sec CNT100 Offset,PR[24:Rotate_Offset] ;
 959:L P[745]  R[157] mm/sec CNT100 Offset,PR[24:Rotate_Offset] ;
 960:L P[746]  R[157] mm/sec CNT100 Offset,PR[24:Rotate_Offset] ;
 961:L P[747]  R[157] mm/sec CNT100 TA    0.00sec,CALL RUN_LASER_STOP Offset,PR[26:Stop_Offset] ;
 963:L P[747]  R[157] mm/sec FINE Offset,PR[76:Offst_dprt] ;
 964:L P[748]  R[157] mm/sec CNT100 Offset,PR[24:Rotate_Offset] ;
 965:L P[749]  R[157] mm/sec CNT100 Offset,PR[24:Rotate_Offset] ;
 966:L P[750]  R[157] mm/sec CNT100 Offset,PR[24:Rotate_Offset] ;
 967:L P[751]  R[157] mm/sec CNT100 Offset,PR[24:Rotate_Offset] ;
 968:L P[752]  R[157] mm/sec CNT100 Offset,PR[24:Rotate_Offset] ;
 969:L P[753]  R[157] mm/sec CNT100 Offset,PR[24:Rotate_Offset] ;
 970: !Pass30 ;
 971: LBL[130:Pass30] ;
 972:L P[754]  R[157] mm/sec FINE Offset,PR[78:Offst_apprch]  ;
 973: WAIT   0.20(sec) ;
 974:L P[754]  R[157] mm/sec CNT100 TA    0.00sec,CALL RUN_LASER_START Offset,PR[25:Start_Offset] ;
 976:L P[755]  R[157] mm/sec CNT100 Offset,PR[24:Rotate_Offset] ;
 977:L P[756]  R[157] mm/sec CNT100 Offset,PR[24:Rotate_Offset] ;
 978:L P[757]  R[157] mm/sec CNT100 Offset,PR[24:Rotate_Offset] ;
 979:L P[758]  R[157] mm/sec CNT100 Offset,PR[24:Rotate_Offset] ;
 980:L P[759]  R[157] mm/sec CNT100 Offset,PR[24:Rotate_Offset] ;
 981:L P[760]  R[157] mm/sec CNT100 Offset,PR[24:Rotate_Offset] ;
 982:L P[761]  R[157] mm/sec CNT100 Offset,PR[24:Rotate_Offset] ;
 983:L P[762]  R[157] mm/sec CNT100 Offset,PR[24:Rotate_Offset] ;
 984:L P[763]  R[157] mm/sec CNT100 Offset,PR[24:Rotate_Offset] ;
 985:L P[764]  R[157] mm/sec CNT100 Offset,PR[24:Rotate_Offset] ;
 986:L P[765]  R[157] mm/sec CNT100 Offset,PR[24:Rotate_Offset] ;
 987:L P[766]  R[157] mm/sec CNT100 TA    0.00sec,CALL RUN_LASER_STOP Offset,PR[26:Stop_Offset] ;
 989:L P[766]  R[157] mm/sec FINE Offset,PR[76:Offst_dprt] ;
 990:L P[767]  R[157] mm/sec CNT100 Offset,PR[24:Rotate_Offset] ;
 991:L P[768]  R[157] mm/sec CNT100 Offset,PR[24:Rotate_Offset] ;
 992:L P[769]  R[157] mm/sec CNT100 Offset,PR[24:Rotate_Offset] ;
 993:L P[770]  R[157] mm/sec CNT100 Offset,PR[24:Rotate_Offset] ;
 994:L P[771]  R[157] mm/sec CNT100 Offset,PR[24:Rotate_Offset] ;
 995:L P[772]  R[157] mm/sec CNT100 Offset,PR[24:Rotate_Offset] ;
 996: !Pass31 ;
 997: LBL[131:Pass31] ;
 998:L P[773]  R[157] mm/sec FINE Offset,PR[78:Offst_apprch]  ;
 999: WAIT   0.20(sec) ;
1000:L P[773]  R[157] mm/sec CNT100 TA    0.00sec,CALL RUN_LASER_START Offset,PR[25:Start_Offset] ;
1002:L P[774]  R[157] mm/sec CNT100 Offset,PR[24:Rotate_Offset] ;
1003:L P[775]  R[157] mm/sec CNT100 Offset,PR[24:Rotate_Offset] ;
1004:L P[776]  R[157] mm/sec CNT100 Offset,PR[24:Rotate_Offset] ;
1005:L P[777]  R[157] mm/sec CNT100 Offset,PR[24:Rotate_Offset] ;
1006:L P[778]  R[157] mm/sec CNT100 Offset,PR[24:Rotate_Offset] ;
1007:L P[779]  R[157] mm/sec CNT100 TA    0.00sec,CALL RUN_LASER_STOP Offset,PR[26:Stop_Offset] ;
1009:L P[779]  R[157] mm/sec FINE Offset,PR[76:Offst_dprt] ;
1010:L P[780]  R[157] mm/sec CNT100 Offset,PR[24:Rotate_Offset] ;
1011:L P[781]  R[157] mm/sec CNT100 Offset,PR[24:Rotate_Offset] ;
1012:L P[782]  R[157] mm/sec CNT100 Offset,PR[24:Rotate_Offset] ;
1013:L P[783]  R[157] mm/sec CNT100 Offset,PR[24:Rotate_Offset] ;
1014:L P[784]  R[157] mm/sec CNT100 Offset,PR[24:Rotate_Offset] ;
1015:L P[785]  R[157] mm/sec CNT100 Offset,PR[24:Rotate_Offset] ;
1016: !Pass32 ;
1017: LBL[132:Pass32] ;
1018:L P[786]  R[157] mm/sec FINE Offset,PR[78:Offst_apprch]  ;
1019: WAIT   0.20(sec) ;
1020:L P[786]  R[157] mm/sec CNT100 TA    0.00sec,CALL RUN_LASER_START Offset,PR[25:Start_Offset] ;
1022:L P[787]  R[157] mm/sec CNT100 Offset,PR[24:Rotate_Offset] ;
1023:L P[788]  R[157] mm/sec CNT100 Offset,PR[24:Rotate_Offset] ;
1024:L P[789]  R[157] mm/sec CNT100 TA    0.00sec,CALL RUN_LASER_STOP Offset,PR[26:Stop_Offset] ;
1026:L P[789]  R[157] mm/sec FINE Offset,PR[76:Offst_dprt] ;
1027:L P[790]  R[157] mm/sec CNT100 Offset,PR[24:Rotate_Offset] ;
1028:L P[791]  R[157] mm/sec CNT100 Offset,PR[24:Rotate_Offset] ;
1029:L P[792]  R[157] mm/sec CNT100 Offset,PR[24:Rotate_Offset] ;
1030:L P[793]  R[157] mm/sec CNT100 Offset,PR[24:Rotate_Offset] ;
1031:L P[794]  R[157] mm/sec CNT100 Offset,PR[24:Rotate_Offset] ;
1032:L P[795]  R[157] mm/sec CNT100 Offset,PR[24:Rotate_Offset] ;
1033: !Pass33 ;
1034: LBL[133:Pass33] ;
1035:L P[796]  R[157] mm/sec FINE Offset,PR[78:Offst_apprch]  ;
1036: WAIT   0.20(sec) ;
1037:L P[796]  R[157] mm/sec CNT100 TA    0.00sec,CALL RUN_LASER_START Offset,PR[25:Start_Offset] ;
1039:L P[797]  R[157] mm/sec CNT100 Offset,PR[24:Rotate_Offset] ;
1040:L P[798]  R[157] mm/sec CNT100 Offset,PR[24:Rotate_Offset] ;
1041:L P[799]  R[157] mm/sec CNT100 TA    0.00sec,CALL RUN_LASER_STOP Offset,PR[26:Stop_Offset] ;
1043:L P[799]  R[157] mm/sec FINE Offset,PR[76:Offst_dprt] ;
1044:L P[800]  R[157] mm/sec CNT100 Offset,PR[24:Rotate_Offset] ;
1045:L P[801]  R[157] mm/sec CNT100 Offset,PR[24:Rotate_Offset] ;
1046:L P[802]  R[157] mm/sec CNT100 Offset,PR[24:Rotate_Offset] ;
1047:L P[803]  R[157] mm/sec CNT100 Offset,PR[24:Rotate_Offset] ;
1048:L P[804]  R[157] mm/sec CNT100 Offset,PR[24:Rotate_Offset] ;
1049:L P[805]  R[157] mm/sec CNT100 Offset,PR[24:Rotate_Offset] ;
1050: !Pass34 ;
1051: LBL[134:Pass34] ;
1052:L P[806]  R[157] mm/sec FINE Offset,PR[78:Offst_apprch]  ;
1053: WAIT   0.20(sec) ;
1054:L P[806]  R[157] mm/sec CNT100 TA    0.00sec,CALL RUN_LASER_START Offset,PR[25:Start_Offset] ;
1056:L P[807]  R[157] mm/sec CNT100 Offset,PR[24:Rotate_Offset] ;
1057:L P[808]  R[157] mm/sec CNT100 Offset,PR[24:Rotate_Offset] ;
1058:L P[809]  R[157] mm/sec CNT100 TA    0.00sec,CALL RUN_LASER_STOP Offset,PR[26:Stop_Offset] ;
1060:L P[809]  R[157] mm/sec FINE Offset,PR[76:Offst_dprt] ;
1061:L P[810]  R[157] mm/sec CNT100 Offset,PR[24:Rotate_Offset] ;
1062:L P[811]  R[157] mm/sec CNT100 Offset,PR[24:Rotate_Offset] ;
1063:L P[812]  R[157] mm/sec CNT100 Offset,PR[24:Rotate_Offset] ;
1064:L P[813]  R[157] mm/sec CNT100 Offset,PR[24:Rotate_Offset] ;
1065:L P[814]  R[157] mm/sec CNT100 Offset,PR[24:Rotate_Offset] ;
1066:L P[815]  R[157] mm/sec CNT100 Offset,PR[24:Rotate_Offset] ;
1067: !Pass35 ;
1068: LBL[135:Pass35] ;
1069:L P[816]  R[157] mm/sec FINE Offset,PR[78:Offst_apprch]  ;
1070: WAIT   0.20(sec) ;
1071:L P[816]  R[157] mm/sec CNT100 TA    0.00sec,CALL RUN_LASER_START Offset,PR[25:Start_Offset] ;
1073:L P[817]  R[157] mm/sec CNT100 Offset,PR[24:Rotate_Offset] ;
1074:L P[818]  R[157] mm/sec CNT100 Offset,PR[24:Rotate_Offset] ;
1075:L P[819]  R[157] mm/sec CNT100 Offset,PR[24:Rotate_Offset] ;
1076:L P[820]  R[157] mm/sec CNT100 Offset,PR[24:Rotate_Offset] ;
1077:L P[821]  R[157] mm/sec CNT100 Offset,PR[24:Rotate_Offset] ;
1078:L P[822]  R[157] mm/sec CNT100 TA    0.00sec,CALL RUN_LASER_STOP Offset,PR[26:Stop_Offset] ;
1080:L P[822]  R[157] mm/sec FINE Offset,PR[76:Offst_dprt] ;
1081:L P[823]  R[157] mm/sec CNT100 Offset,PR[24:Rotate_Offset] ;
1082:L P[824]  R[157] mm/sec CNT100 Offset,PR[24:Rotate_Offset] ;
1083:L P[825]  R[157] mm/sec CNT100 Offset,PR[24:Rotate_Offset] ;
1084:L P[826]  R[157] mm/sec CNT100 Offset,PR[24:Rotate_Offset] ;
1085:L P[827]  R[157] mm/sec CNT100 Offset,PR[24:Rotate_Offset] ;
1086:L P[828]  R[157] mm/sec CNT100 Offset,PR[24:Rotate_Offset] ;
1087: !Pass36 ;
1088: LBL[136:Pass36] ;
1089:L P[829]  R[157] mm/sec FINE Offset,PR[78:Offst_apprch]  ;
1090: WAIT   0.20(sec) ;
1091:L P[829]  R[157] mm/sec CNT100 TA    0.00sec,CALL RUN_LASER_START Offset,PR[25:Start_Offset] ;
1093:L P[830]  R[157] mm/sec CNT100 Offset,PR[24:Rotate_Offset] ;
1094:L P[831]  R[157] mm/sec CNT100 Offset,PR[24:Rotate_Offset] ;
1095:L P[832]  R[157] mm/sec CNT100 TA    0.00sec,CALL RUN_LASER_STOP Offset,PR[26:Stop_Offset] ;
1097:L P[832]  R[157] mm/sec FINE Offset,PR[76:Offst_dprt] ;
1098:L P[833]  R[157] mm/sec CNT100 Offset,PR[24:Rotate_Offset] ;
1099:L P[834]  R[157] mm/sec CNT100 Offset,PR[24:Rotate_Offset] ;
1100:L P[835]  R[157] mm/sec CNT100 Offset,PR[24:Rotate_Offset] ;
1101:L P[836]  R[157] mm/sec CNT100 Offset,PR[24:Rotate_Offset] ;
1102:L P[837]  R[157] mm/sec CNT100 Offset,PR[24:Rotate_Offset] ;
1103:L P[838]  R[157] mm/sec CNT100 Offset,PR[24:Rotate_Offset] ;
1104: !Pass37 ;
1105: LBL[137:Pass37] ;
1106:L P[839]  R[157] mm/sec FINE Offset,PR[78:Offst_apprch]  ;
1107: WAIT   0.20(sec) ;
1108:L P[839]  R[157] mm/sec CNT100 TA    0.00sec,CALL RUN_LASER_START Offset,PR[25:Start_Offset] ;
1110:L P[840]  R[157] mm/sec CNT100 Offset,PR[24:Rotate_Offset] ;
1111:L P[841]  R[157] mm/sec CNT100 Offset,PR[24:Rotate_Offset] ;
1112:L P[842]  R[157] mm/sec CNT100 TA    0.00sec,CALL RUN_LASER_STOP Offset,PR[26:Stop_Offset] ;
1114:L P[842]  R[157] mm/sec FINE Offset,PR[76:Offst_dprt] ;
1115:L P[843]  R[157] mm/sec CNT100 Offset,PR[24:Rotate_Offset] ;
1116:L P[844]  R[157] mm/sec CNT100 Offset,PR[24:Rotate_Offset] ;
1117:L P[845]  R[157] mm/sec CNT100 Offset,PR[24:Rotate_Offset] ;
1118:L P[846]  R[157] mm/sec CNT100 Offset,PR[24:Rotate_Offset] ;
1119:L P[847]  R[157] mm/sec CNT100 Offset,PR[24:Rotate_Offset] ;
1120:L P[848]  R[157] mm/sec CNT100 Offset,PR[24:Rotate_Offset] ;
1121: !Pass38 ;
1122: LBL[138:Pass38] ;
1123:L P[849]  R[157] mm/sec FINE Offset,PR[78:Offst_apprch]  ;
1124: WAIT   0.20(sec) ;
1125:L P[849]  R[157] mm/sec CNT100 TA    0.00sec,CALL RUN_LASER_START Offset,PR[25:Start_Offset] ;
1127:L P[850]  R[157] mm/sec CNT100 Offset,PR[24:Rotate_Offset] ;
1128:L P[851]  R[157] mm/sec CNT100 Offset,PR[24:Rotate_Offset] ;
1129:L P[852]  R[157] mm/sec CNT100 TA    0.00sec,CALL RUN_LASER_STOP Offset,PR[26:Stop_Offset] ;
1131:L P[852]  R[157] mm/sec FINE Offset,PR[76:Offst_dprt] ;
1132:L P[853]  R[157] mm/sec CNT100 Offset,PR[24:Rotate_Offset] ;
1133:L P[854]  R[157] mm/sec CNT100 Offset,PR[24:Rotate_Offset] ;
1134:L P[855]  R[157] mm/sec CNT100 Offset,PR[24:Rotate_Offset] ;
1135:L P[856]  R[157] mm/sec CNT100 Offset,PR[24:Rotate_Offset] ;
1136:L P[857]  R[157] mm/sec CNT100 Offset,PR[24:Rotate_Offset] ;
1137:L P[858]  R[157] mm/sec CNT100 Offset,PR[24:Rotate_Offset] ;
1138: !Pass39 ;
1139: LBL[139:Pass39] ;
1140:L P[859]  R[157] mm/sec FINE Offset,PR[78:Offst_apprch]  ;
1141: WAIT   0.20(sec) ;
1142:L P[859]  R[157] mm/sec CNT100 TA    0.00sec,CALL RUN_LASER_START Offset,PR[25:Start_Offset] ;
1144:L P[860]  R[157] mm/sec CNT100 Offset,PR[24:Rotate_Offset] ;
1145:L P[861]  R[157] mm/sec CNT100 Offset,PR[24:Rotate_Offset] ;
1146:L P[862]  R[157] mm/sec CNT100 TA    0.00sec,CALL RUN_LASER_STOP Offset,PR[26:Stop_Offset] ;
1148:L P[862]  R[157] mm/sec FINE Offset,PR[76:Offst_dprt] ;
1149:L P[863]  R[157] mm/sec CNT100 Offset,PR[24:Rotate_Offset] ;
1150:L P[864]  R[157] mm/sec CNT100 Offset,PR[24:Rotate_Offset] ;
1151:L P[865]  R[157] mm/sec CNT100 Offset,PR[24:Rotate_Offset] ;
1152:L P[866]  R[157] mm/sec CNT100 Offset,PR[24:Rotate_Offset] ;
1153:L P[867]  R[157] mm/sec CNT100 Offset,PR[24:Rotate_Offset] ;
1154:L P[868]  R[157] mm/sec CNT100 Offset,PR[24:Rotate_Offset] ;
1155: !Pass40 ;
1156: LBL[140:Pass40] ;
1157:L P[869]  R[157] mm/sec FINE Offset,PR[78:Offst_apprch]  ;
1158: WAIT   0.20(sec) ;
1159:L P[869]  R[157] mm/sec CNT100 TA    0.00sec,CALL RUN_LASER_START Offset,PR[25:Start_Offset] ;
1161:L P[870]  R[157] mm/sec CNT100 Offset,PR[24:Rotate_Offset] ;
1162:L P[871]  R[157] mm/sec CNT100 Offset,PR[24:Rotate_Offset] ;
1163:L P[872]  R[157] mm/sec CNT100 Offset,PR[24:Rotate_Offset] ;
1164:L P[873]  R[157] mm/sec CNT100 Offset,PR[24:Rotate_Offset] ;
1165:L P[874]  R[157] mm/sec CNT100 Offset,PR[24:Rotate_Offset] ;
1166:L P[875]  R[157] mm/sec CNT100 Offset,PR[24:Rotate_Offset] ;
1167:L P[876]  R[157] mm/sec CNT100 Offset,PR[24:Rotate_Offset] ;
1168:L P[877]  R[157] mm/sec CNT100 TA    0.00sec,CALL RUN_LASER_STOP Offset,PR[26:Stop_Offset] ;
1170:L P[877]  R[157] mm/sec FINE Offset,PR[76:Offst_dprt] ;
1171:L P[878]  R[157] mm/sec CNT100 Offset,PR[24:Rotate_Offset] ;
1172:L P[879]  R[157] mm/sec CNT100 Offset,PR[24:Rotate_Offset] ;
1173:L P[880]  R[157] mm/sec CNT100 Offset,PR[24:Rotate_Offset] ;
1174:L P[881]  R[157] mm/sec CNT100 Offset,PR[24:Rotate_Offset] ;
1175:L P[882]  R[157] mm/sec CNT100 Offset,PR[24:Rotate_Offset] ;
1176:L P[883]  R[157] mm/sec CNT100 Offset,PR[24:Rotate_Offset] ;
1177: !Pass41 ;
1178: LBL[141:Pass41] ;
1179:L P[884]  R[157] mm/sec FINE Offset,PR[78:Offst_apprch]  ;
1180: WAIT   0.20(sec) ;
1181:L P[884]  R[157] mm/sec CNT100 TA    0.00sec,CALL RUN_LASER_START Offset,PR[25:Start_Offset] ;
1183:L P[885]  R[157] mm/sec CNT100 Offset,PR[24:Rotate_Offset] ;
1184:L P[886]  R[157] mm/sec CNT100 Offset,PR[24:Rotate_Offset] ;
1185:L P[887]  R[157] mm/sec CNT100 Offset,PR[24:Rotate_Offset] ;
1186:L P[888]  R[157] mm/sec CNT100 Offset,PR[24:Rotate_Offset] ;
1187:L P[889]  R[157] mm/sec CNT100 TA    0.00sec,CALL RUN_LASER_STOP Offset,PR[26:Stop_Offset] ;
1189:L P[889]  R[157] mm/sec FINE Offset,PR[76:Offst_dprt] ;
1190:L P[890]  R[157] mm/sec CNT100 Offset,PR[24:Rotate_Offset] ;
1191:L P[891]  R[157] mm/sec CNT100 Offset,PR[24:Rotate_Offset] ;
1192:L P[892]  R[157] mm/sec CNT100 Offset,PR[24:Rotate_Offset] ;
1193:L P[893]  R[157] mm/sec CNT100 Offset,PR[24:Rotate_Offset] ;
1194:L P[894]  R[157] mm/sec CNT100 Offset,PR[24:Rotate_Offset] ;
1195:L P[895]  R[157] mm/sec CNT100 Offset,PR[24:Rotate_Offset] ;
1196: !Pass42 ;
1197: LBL[142:Pass42] ;
1198:L P[896]  R[157] mm/sec FINE Offset,PR[78:Offst_apprch]  ;
1199: WAIT   0.20(sec) ;
1200:L P[896]  R[157] mm/sec CNT100 TA    0.00sec,CALL RUN_LASER_START Offset,PR[25:Start_Offset] ;
1202:L P[897]  R[157] mm/sec CNT100 Offset,PR[24:Rotate_Offset] ;
1203:L P[898]  R[157] mm/sec CNT100 Offset,PR[24:Rotate_Offset] ;
1204:L P[899]  R[157] mm/sec CNT100 Offset,PR[24:Rotate_Offset] ;
1205:L P[900]  R[157] mm/sec CNT100 Offset,PR[24:Rotate_Offset] ;
1206:L P[901]  R[157] mm/sec CNT100 Offset,PR[24:Rotate_Offset] ;
1207:L P[902]  R[157] mm/sec CNT100 TA    0.00sec,CALL RUN_LASER_STOP Offset,PR[26:Stop_Offset] ;
1209:L P[902]  R[157] mm/sec FINE Offset,PR[76:Offst_dprt] ;
1210:L P[903]  R[157] mm/sec CNT100 Offset,PR[24:Rotate_Offset] ;
1211:L P[904]  R[157] mm/sec CNT100 Offset,PR[24:Rotate_Offset] ;
1212:L P[905]  R[157] mm/sec CNT100 Offset,PR[24:Rotate_Offset] ;
1213:L P[906]  R[157] mm/sec CNT100 Offset,PR[24:Rotate_Offset] ;
1214:L P[907]  R[157] mm/sec CNT100 Offset,PR[24:Rotate_Offset] ;
1215:L P[908]  R[157] mm/sec CNT100 Offset,PR[24:Rotate_Offset] ;
1216: !Pass43 ;
1217: LBL[143:Pass43] ;
1218:L P[909]  R[157] mm/sec FINE Offset,PR[78:Offst_apprch]  ;
1219: WAIT   0.20(sec) ;
1220:L P[909]  R[157] mm/sec CNT100 TA    0.00sec,CALL RUN_LASER_START Offset,PR[25:Start_Offset] ;
1222:L P[910]  R[157] mm/sec CNT100 Offset,PR[24:Rotate_Offset] ;
1223:L P[911]  R[157] mm/sec CNT100 Offset,PR[24:Rotate_Offset] ;
1224:L P[912]  R[157] mm/sec CNT100 TA    0.00sec,CALL RUN_LASER_STOP Offset,PR[26:Stop_Offset] ;
1226:L P[912]  R[157] mm/sec FINE Offset,PR[76:Offst_dprt] ;
1227:L P[913]  R[157] mm/sec CNT100 Offset,PR[24:Rotate_Offset] ;
1228:L P[914]  R[157] mm/sec CNT100 Offset,PR[24:Rotate_Offset] ;
1229:L P[915]  R[157] mm/sec CNT100 Offset,PR[24:Rotate_Offset] ;
1230:L P[916]  R[157] mm/sec CNT100 Offset,PR[24:Rotate_Offset] ;
1231:L P[917]  R[157] mm/sec CNT100 Offset,PR[24:Rotate_Offset] ;
1232:L P[918]  R[157] mm/sec CNT100 Offset,PR[24:Rotate_Offset] ;
1233: !Pass44 ;
1234: LBL[144:Pass44] ;
1235:L P[919]  R[157] mm/sec FINE Offset,PR[78:Offst_apprch]  ;
1236: WAIT   0.20(sec) ;
1237:L P[919]  R[157] mm/sec CNT100 TA    0.00sec,CALL RUN_LASER_START Offset,PR[25:Start_Offset] ;
1239:L P[920]  R[157] mm/sec CNT100 Offset,PR[24:Rotate_Offset] ;
1240:L P[921]  R[157] mm/sec CNT100 Offset,PR[24:Rotate_Offset] ;
1241:L P[922]  R[157] mm/sec CNT100 TA    0.00sec,CALL RUN_LASER_STOP Offset,PR[26:Stop_Offset] ;
1243:L P[922]  R[157] mm/sec FINE Offset,PR[76:Offst_dprt] ;
1244:L P[923]  R[157] mm/sec CNT100 Offset,PR[24:Rotate_Offset] ;
1245:L P[924]  R[157] mm/sec CNT100 Offset,PR[24:Rotate_Offset] ;
1246:L P[925]  R[157] mm/sec CNT100 Offset,PR[24:Rotate_Offset] ;
1247:L P[926]  R[157] mm/sec CNT100 Offset,PR[24:Rotate_Offset] ;
1248:L P[927]  R[157] mm/sec CNT100 Offset,PR[24:Rotate_Offset] ;
1249:L P[928]  R[157] mm/sec CNT100 Offset,PR[24:Rotate_Offset] ;
1250: !Pass45 ;
1251: LBL[145:Pass45] ;
1252:L P[929]  R[157] mm/sec FINE Offset,PR[78:Offst_apprch]  ;
1253: WAIT   0.20(sec) ;
1254:L P[929]  R[157] mm/sec CNT100 TA    0.00sec,CALL RUN_LASER_START Offset,PR[25:Start_Offset] ;
1256:L P[930]  R[157] mm/sec CNT100 Offset,PR[24:Rotate_Offset] ;
1257:L P[931]  R[157] mm/sec CNT100 Offset,PR[24:Rotate_Offset] ;
1258:L P[932]  R[157] mm/sec CNT100 Offset,PR[24:Rotate_Offset] ;
1259:L P[933]  R[157] mm/sec CNT100 TA    0.00sec,CALL RUN_LASER_STOP Offset,PR[26:Stop_Offset] ;
1261:L P[933]  R[157] mm/sec FINE Offset,PR[76:Offst_dprt] ;
1262:L P[934]  R[157] mm/sec CNT100 Offset,PR[24:Rotate_Offset] ;
1263:L P[935]  R[157] mm/sec CNT100 Offset,PR[24:Rotate_Offset] ;
1264:L P[936]  R[157] mm/sec CNT100 Offset,PR[24:Rotate_Offset] ;
1265:L P[937]  R[157] mm/sec CNT100 Offset,PR[24:Rotate_Offset] ;
1266:L P[938]  R[157] mm/sec CNT100 Offset,PR[24:Rotate_Offset] ;
1267:L P[939]  R[157] mm/sec CNT100 Offset,PR[24:Rotate_Offset] ;
1268: !Pass46 ;
1269: LBL[146:Pass46] ;
1270:L P[940]  R[157] mm/sec FINE Offset,PR[78:Offst_apprch]  ;
1271: WAIT   0.20(sec) ;
1272:L P[940]  R[157] mm/sec CNT100 TA    0.00sec,CALL RUN_LASER_START Offset,PR[25:Start_Offset] ;
1274:L P[941]  R[157] mm/sec CNT100 Offset,PR[24:Rotate_Offset] ;
1275:L P[942]  R[157] mm/sec CNT100 Offset,PR[24:Rotate_Offset] ;
1276:L P[943]  R[157] mm/sec CNT100 Offset,PR[24:Rotate_Offset] ;
1277:L P[944]  R[157] mm/sec CNT100 TA    0.00sec,CALL RUN_LASER_STOP Offset,PR[26:Stop_Offset] ;
1279:L P[944]  R[157] mm/sec FINE Offset,PR[76:Offst_dprt] ;
1280:L P[945]  R[157] mm/sec CNT100 Offset,PR[24:Rotate_Offset] ;
1281:L P[946]  R[157] mm/sec CNT100 Offset,PR[24:Rotate_Offset] ;
1282:L P[947]  R[157] mm/sec CNT100 Offset,PR[24:Rotate_Offset] ;
1283:L P[948]  R[157] mm/sec CNT100 Offset,PR[24:Rotate_Offset] ;
1284:L P[949]  R[157] mm/sec CNT100 Offset,PR[24:Rotate_Offset] ;
1285:L P[950]  R[157] mm/sec CNT100 Offset,PR[24:Rotate_Offset] ;
1286: !Pass47 ;
1287: LBL[147:Pass47] ;
1288:L P[951]  R[157] mm/sec FINE Offset,PR[78:Offst_apprch]  ;
1289: WAIT   0.20(sec) ;
1290:L P[951]  R[157] mm/sec CNT100 TA    0.00sec,CALL RUN_LASER_START Offset,PR[25:Start_Offset] ;
1292:L P[952]  R[157] mm/sec CNT100 Offset,PR[24:Rotate_Offset] ;
1293:L P[953]  R[157] mm/sec CNT100 Offset,PR[24:Rotate_Offset] ;
1294:L P[954]  R[157] mm/sec CNT100 Offset,PR[24:Rotate_Offset] ;
1295:L P[955]  R[157] mm/sec CNT100 Offset,PR[24:Rotate_Offset] ;
1296:L P[956]  R[157] mm/sec CNT100 Offset,PR[24:Rotate_Offset] ;
1297:L P[957]  R[157] mm/sec CNT100 TA    0.00sec,CALL RUN_LASER_STOP Offset,PR[26:Stop_Offset] ;
1299:L P[957]  R[157] mm/sec FINE Offset,PR[76:Offst_dprt] ;
1300:L P[958]  R[157] mm/sec CNT100 Offset,PR[24:Rotate_Offset] ;
1301:L P[959]  R[157] mm/sec CNT100 Offset,PR[24:Rotate_Offset] ;
1302:L P[960]  R[157] mm/sec CNT100 Offset,PR[24:Rotate_Offset] ;
1303:L P[961]  R[157] mm/sec CNT100 Offset,PR[24:Rotate_Offset] ;
1304:L P[962]  R[157] mm/sec CNT100 Offset,PR[24:Rotate_Offset] ;
1305:L P[963]  R[157] mm/sec CNT100 Offset,PR[24:Rotate_Offset] ;
1306: !Pass48 ;
1307: LBL[148:Pass48] ;
1308:L P[964]  R[157] mm/sec FINE Offset,PR[78:Offst_apprch]  ;
1309: WAIT   0.20(sec) ;
1310:L P[964]  R[157] mm/sec CNT100 TA    0.00sec,CALL RUN_LASER_START Offset,PR[25:Start_Offset] ;
1312:L P[965]  R[157] mm/sec CNT100 Offset,PR[24:Rotate_Offset] ;
1313:L P[966]  R[157] mm/sec CNT100 TA    0.00sec,CALL RUN_LASER_STOP Offset,PR[26:Stop_Offset] ;
1315:L P[966]  R[157] mm/sec FINE Offset,PR[76:Offst_dprt] ;
1316:L P[967]  R[157] mm/sec CNT100 Offset,PR[24:Rotate_Offset] ;
1317:L P[968]  R[157] mm/sec CNT100 Offset,PR[24:Rotate_Offset] ;
1318:L P[969]  R[157] mm/sec CNT100 Offset,PR[24:Rotate_Offset] ;
1319:L P[970]  R[157] mm/sec CNT100 Offset,PR[24:Rotate_Offset] ;
1320:L P[971]  R[157] mm/sec CNT100 Offset,PR[24:Rotate_Offset] ;
1321:L P[972]  R[157] mm/sec CNT100 Offset,PR[24:Rotate_Offset] ;
1322: !Pass49 ;
1323: LBL[149:Pass49] ;
1324:L P[973]  R[157] mm/sec FINE Offset,PR[78:Offst_apprch]  ;
1325: WAIT   0.20(sec) ;
1326:L P[973]  R[157] mm/sec CNT100 TA    0.00sec,CALL RUN_LASER_START Offset,PR[25:Start_Offset] ;
1328:L P[974]  R[157] mm/sec CNT100 Offset,PR[24:Rotate_Offset] ;
1329:L P[975]  R[157] mm/sec CNT100 TA    0.00sec,CALL RUN_LASER_STOP Offset,PR[26:Stop_Offset] ;
1331:L P[975]  R[157] mm/sec FINE Offset,PR[76:Offst_dprt] ;
1332:L P[976]  R[157] mm/sec CNT100 Offset,PR[24:Rotate_Offset] ;
1333:L P[977]  R[157] mm/sec CNT100 Offset,PR[24:Rotate_Offset] ;
1334:L P[978]  R[157] mm/sec CNT100 Offset,PR[24:Rotate_Offset] ;
1335:L P[979]  R[157] mm/sec CNT100 Offset,PR[24:Rotate_Offset] ;
1336:L P[980]  R[157] mm/sec CNT100 Offset,PR[24:Rotate_Offset] ;
1337:L P[981]  R[157] mm/sec CNT100 Offset,PR[24:Rotate_Offset] ;
1338: !Pass50 ;
1339: LBL[150:Pass50] ;
1340:L P[982]  R[157] mm/sec FINE Offset,PR[78:Offst_apprch]  ;
1341: WAIT   0.20(sec) ;
1342:L P[982]  R[157] mm/sec CNT100 TA    0.00sec,CALL RUN_LASER_START Offset,PR[25:Start_Offset] ;
1344:L P[983]  R[157] mm/sec CNT100 Offset,PR[24:Rotate_Offset] ;
1345:L P[984]  R[157] mm/sec CNT100 TA    0.00sec,CALL RUN_LASER_STOP Offset,PR[26:Stop_Offset] ;
1347:L P[984]  R[157] mm/sec FINE Offset,PR[76:Offst_dprt] ;
1348:L P[985]  R[157] mm/sec CNT100 Offset,PR[24:Rotate_Offset] ;
1349:L P[986]  R[157] mm/sec CNT100 Offset,PR[24:Rotate_Offset] ;
1350:L P[987]  R[157] mm/sec CNT100 Offset,PR[24:Rotate_Offset] ;
1351:L P[988]  R[157] mm/sec CNT100 Offset,PR[24:Rotate_Offset] ;
1352:L P[989]  R[157] mm/sec CNT100 Offset,PR[24:Rotate_Offset] ;
1353:L P[990]  R[157] mm/sec CNT100 Offset,PR[24:Rotate_Offset] ;
1354: !Pass51 ;
1355: LBL[151:Pass51] ;
1356:L P[991]  R[157] mm/sec FINE Offset,PR[78:Offst_apprch]  ;
1357: WAIT   0.20(sec) ;
1358:L P[991]  R[157] mm/sec CNT100 TA    0.00sec,CALL RUN_LASER_START Offset,PR[25:Start_Offset] ;
1360:L P[992]  R[157] mm/sec CNT100 Offset,PR[24:Rotate_Offset] ;
1361:L P[993]  R[157] mm/sec CNT100 TA    0.00sec,CALL RUN_LASER_STOP Offset,PR[26:Stop_Offset] ;
1363:L P[993]  R[157] mm/sec FINE Offset,PR[76:Offst_dprt] ;
1364:L P[994]  R[157] mm/sec CNT100 Offset,PR[24:Rotate_Offset] ;
1365:L P[995]  R[157] mm/sec CNT100 Offset,PR[24:Rotate_Offset] ;
1366:L P[996]  R[157] mm/sec CNT100 Offset,PR[24:Rotate_Offset] ;
1367:L P[997]  R[157] mm/sec CNT100 Offset,PR[24:Rotate_Offset] ;
1368:L P[998]  R[157] mm/sec CNT100 Offset,PR[24:Rotate_Offset] ;
1369:L P[999]  R[157] mm/sec CNT100 Offset,PR[24:Rotate_Offset] ;
1370: !Pass52 ;
1371: LBL[152:Pass52] ;
1372:L P[1000]  R[157] mm/sec FINE Offset,PR[78:Offst_apprch]  ;
1373: WAIT   0.20(sec) ;
1374:L P[1000]  R[157] mm/sec CNT100 TA    0.00sec,CALL RUN_LASER_START Offset,PR[25:Start_Offset] ;
1376:L P[1001]  R[157] mm/sec CNT100 Offset,PR[24:Rotate_Offset] ;
1377:L P[1002]  R[157] mm/sec CNT100 Offset,PR[24:Rotate_Offset] ;
1378:L P[1003]  R[157] mm/sec CNT100 Offset,PR[24:Rotate_Offset] ;
1379:L P[1004]  R[157] mm/sec CNT100 Offset,PR[24:Rotate_Offset] ;
1380:L P[1005]  R[157] mm/sec CNT100 Offset,PR[24:Rotate_Offset] ;
1381:L P[1006]  R[157] mm/sec CNT100 TA    0.00sec,CALL RUN_LASER_STOP Offset,PR[26:Stop_Offset] ;
1383:L P[1006]  R[157] mm/sec FINE Offset,PR[76:Offst_dprt] ;
1384:L P[1007]  R[157] mm/sec CNT100 Offset,PR[24:Rotate_Offset] ;
1385:L P[1008]  R[157] mm/sec CNT100 Offset,PR[24:Rotate_Offset] ;
1386:L P[1009]  R[157] mm/sec CNT100 Offset,PR[24:Rotate_Offset] ;
1387:L P[1010]  R[157] mm/sec CNT100 Offset,PR[24:Rotate_Offset] ;
1388:L P[1011]  R[157] mm/sec CNT100 Offset,PR[24:Rotate_Offset] ;
1389:L P[1012]  R[157] mm/sec CNT100 Offset,PR[24:Rotate_Offset] ;
1390: !Pass53 ;
1391: LBL[153:Pass53] ;
1392:L P[1013]  R[157] mm/sec FINE Offset,PR[78:Offst_apprch]  ;
1393: WAIT   0.20(sec) ;
1394:L P[1013]  R[157] mm/sec CNT100 TA    0.00sec,CALL RUN_LASER_START Offset,PR[25:Start_Offset] ;
1396:L P[1014]  R[157] mm/sec CNT100 Offset,PR[24:Rotate_Offset] ;
1397:L P[1015]  R[157] mm/sec CNT100 TA    0.00sec,CALL RUN_LASER_STOP Offset,PR[26:Stop_Offset] ;
1399:L P[1015]  R[157] mm/sec FINE Offset,PR[76:Offst_dprt] ;
1400:L P[1016]  R[157] mm/sec CNT100 Offset,PR[24:Rotate_Offset] ;
1401:L P[1017]  R[157] mm/sec CNT100 Offset,PR[24:Rotate_Offset] ;
1402:L P[1018]  R[157] mm/sec CNT100 Offset,PR[24:Rotate_Offset] ;
1403:L P[1019]  R[157] mm/sec CNT100 Offset,PR[24:Rotate_Offset] ;
1404:L P[1020]  R[157] mm/sec CNT100 Offset,PR[24:Rotate_Offset] ;
1405:L P[1021]  R[157] mm/sec CNT100 Offset,PR[24:Rotate_Offset] ;
1406: !Pass54 ;
1407: LBL[154:Pass54] ;
1408:L P[1022]  R[157] mm/sec FINE Offset,PR[78:Offst_apprch]  ;
1409: WAIT   0.20(sec) ;
1410:L P[1022]  R[157] mm/sec CNT100 TA    0.00sec,CALL RUN_LASER_START Offset,PR[25:Start_Offset] ;
1412:L P[1023]  R[157] mm/sec CNT100 Offset,PR[24:Rotate_Offset] ;
1413:L P[1024]  R[157] mm/sec CNT100 Offset,PR[24:Rotate_Offset] ;
1414:L P[1025]  R[157] mm/sec CNT100 TA    0.00sec,CALL RUN_LASER_STOP Offset,PR[26:Stop_Offset] ;
1416:L P[1025]  R[157] mm/sec FINE Offset,PR[76:Offst_dprt] ;
1417:L P[1026]  R[157] mm/sec CNT100 Offset,PR[24:Rotate_Offset] ;
1418:L P[1027]  R[157] mm/sec CNT100 Offset,PR[24:Rotate_Offset] ;
1419:L P[1028]  R[157] mm/sec CNT100 Offset,PR[24:Rotate_Offset] ;
1420:L P[1029]  R[157] mm/sec CNT100 Offset,PR[24:Rotate_Offset] ;
1421:L P[1030]  R[157] mm/sec CNT100 Offset,PR[24:Rotate_Offset] ;
1422:L P[1031]  R[157] mm/sec CNT100 Offset,PR[24:Rotate_Offset] ;
1423: !Pass55 ;
1424: LBL[155:Pass55] ;
1425:L P[1032]  R[157] mm/sec FINE Offset,PR[78:Offst_apprch]  ;
1426: WAIT   0.20(sec) ;
1427:L P[1032]  R[157] mm/sec CNT100 TA    0.00sec,CALL RUN_LASER_START Offset,PR[25:Start_Offset] ;
1429:L P[1033]  R[157] mm/sec CNT100 Offset,PR[24:Rotate_Offset] ;
1430:L P[1034]  R[157] mm/sec CNT100 Offset,PR[24:Rotate_Offset] ;
1431:L P[1035]  R[157] mm/sec CNT100 TA    0.00sec,CALL RUN_LASER_STOP Offset,PR[26:Stop_Offset] ;
1433:L P[1035]  R[157] mm/sec FINE Offset,PR[76:Offst_dprt] ;
1434:L P[1036]  R[157] mm/sec CNT100 Offset,PR[24:Rotate_Offset] ;
1435:L P[1037]  R[157] mm/sec CNT100 Offset,PR[24:Rotate_Offset] ;
1436:L P[1038]  R[157] mm/sec CNT100 Offset,PR[24:Rotate_Offset] ;
1437:L P[1039]  R[157] mm/sec CNT100 Offset,PR[24:Rotate_Offset] ;
1438:L P[1040]  R[157] mm/sec CNT100 Offset,PR[24:Rotate_Offset] ;
1439:L P[1041]  R[157] mm/sec CNT100 Offset,PR[24:Rotate_Offset] ;
1440: !Pass56 ;
1441: LBL[156:Pass56] ;
1442:L P[1042]  R[157] mm/sec FINE Offset,PR[78:Offst_apprch]  ;
1443: WAIT   0.20(sec) ;
1444:L P[1042]  R[157] mm/sec CNT100 TA    0.00sec,CALL RUN_LASER_START Offset,PR[25:Start_Offset] ;
1446:L P[1043]  R[157] mm/sec CNT100 Offset,PR[24:Rotate_Offset] ;
1447:L P[1044]  R[157] mm/sec CNT100 Offset,PR[24:Rotate_Offset] ;
1448:L P[1045]  R[157] mm/sec CNT100 TA    0.00sec,CALL RUN_LASER_STOP Offset,PR[26:Stop_Offset] ;
1450:L P[1045]  R[157] mm/sec FINE Offset,PR[76:Offst_dprt] ;
1451:L P[1046]  R[157] mm/sec CNT100 Offset,PR[24:Rotate_Offset] ;
1452:L P[1047]  R[157] mm/sec CNT100 Offset,PR[24:Rotate_Offset] ;
1453:L P[1048]  R[157] mm/sec CNT100 Offset,PR[24:Rotate_Offset] ;
1454:L P[1049]  R[157] mm/sec CNT100 Offset,PR[24:Rotate_Offset] ;
1455:L P[1050]  R[157] mm/sec CNT100 Offset,PR[24:Rotate_Offset] ;
1456:L P[1051]  R[157] mm/sec CNT100 Offset,PR[24:Rotate_Offset] ;
1457: !Pass57 ;
1458: LBL[157:Pass57] ;
1459:L P[1052]  R[157] mm/sec FINE Offset,PR[78:Offst_apprch]  ;
1460: WAIT   0.20(sec) ;
1461:L P[1052]  R[157] mm/sec CNT100 TA    0.00sec,CALL RUN_LASER_START Offset,PR[25:Start_Offset] ;
1463:L P[1053]  R[157] mm/sec CNT100 Offset,PR[24:Rotate_Offset] ;
1464:L P[1054]  R[157] mm/sec CNT100 TA    0.00sec,CALL RUN_LASER_STOP Offset,PR[26:Stop_Offset] ;
1466:L P[1054]  R[157] mm/sec FINE Offset,PR[76:Offst_dprt] ;
1467:L P[1055]  R[157] mm/sec CNT100 Offset,PR[24:Rotate_Offset] ;
1468:L P[1056]  R[157] mm/sec CNT100 Offset,PR[24:Rotate_Offset] ;
1469:L P[1057]  R[157] mm/sec CNT100 Offset,PR[24:Rotate_Offset] ;
1470:L P[1058]  R[157] mm/sec CNT100 Offset,PR[24:Rotate_Offset] ;
1471:L P[1059]  R[157] mm/sec CNT100 Offset,PR[24:Rotate_Offset] ;
1472:L P[1060]  R[157] mm/sec CNT100 Offset,PR[24:Rotate_Offset] ;
1473: !Pass58 ;
1474: LBL[158:Pass58] ;
1475:L P[1061]  R[157] mm/sec FINE Offset,PR[78:Offst_apprch]  ;
1476: WAIT   0.20(sec) ;
1477:L P[1061]  R[157] mm/sec CNT100 TA    0.00sec,CALL RUN_LASER_START Offset,PR[25:Start_Offset] ;
1479:L P[1062]  R[157] mm/sec CNT100 Offset,PR[24:Rotate_Offset] ;
1480:L P[1063]  R[157] mm/sec CNT100 TA    0.00sec,CALL RUN_LASER_STOP Offset,PR[26:Stop_Offset] ;
1482:L P[1063]  R[157] mm/sec FINE Offset,PR[76:Offst_dprt] ;
1483:L P[1064]  R[157] mm/sec CNT100 Offset,PR[24:Rotate_Offset] ;
1484:L P[1065]  R[157] mm/sec CNT100 Offset,PR[24:Rotate_Offset] ;
1485:L P[1066]  R[157] mm/sec CNT100 Offset,PR[24:Rotate_Offset] ;
1486:L P[1067]  R[157] mm/sec CNT100 Offset,PR[24:Rotate_Offset] ;
1487:L P[1068]  R[157] mm/sec CNT100 Offset,PR[24:Rotate_Offset] ;
1488:L P[1069]  R[157] mm/sec CNT100 Offset,PR[24:Rotate_Offset] ;
1489: !Pass59 ;
1490: LBL[159:Pass59] ;
1491:L P[1070]  R[157] mm/sec FINE Offset,PR[78:Offst_apprch]  ;
1492: WAIT   0.20(sec) ;
1493:L P[1070]  R[157] mm/sec CNT100 TA    0.00sec,CALL RUN_LASER_START Offset,PR[25:Start_Offset] ;
1495:L P[1071]  R[157] mm/sec CNT100 Offset,PR[24:Rotate_Offset] ;
1496:L P[1072]  R[157] mm/sec CNT100 Offset,PR[24:Rotate_Offset] ;
1497:L P[1073]  R[157] mm/sec CNT100 Offset,PR[24:Rotate_Offset] ;
1498:L P[1074]  R[157] mm/sec CNT100 Offset,PR[24:Rotate_Offset] ;
1499:L P[1075]  R[157] mm/sec CNT100 TA    0.00sec,CALL RUN_LASER_STOP Offset,PR[26:Stop_Offset] ;
1501:L P[1075]  R[157] mm/sec FINE Offset,PR[76:Offst_dprt] ;
1502:L P[1076]  R[157] mm/sec CNT100 Offset,PR[24:Rotate_Offset] ;
1503:L P[1077]  R[157] mm/sec CNT100 Offset,PR[24:Rotate_Offset] ;
1504:L P[1078]  R[157] mm/sec CNT100 Offset,PR[24:Rotate_Offset] ;
1505:L P[1079]  R[157] mm/sec CNT100 Offset,PR[24:Rotate_Offset] ;
1506:L P[1080]  R[157] mm/sec CNT100 Offset,PR[24:Rotate_Offset] ;
1507:L P[1081]  R[157] mm/sec CNT100 Offset,PR[24:Rotate_Offset] ;
1508: !Pass60 ;
1509: LBL[160:Pass60] ;
1510:L P[1082]  R[157] mm/sec FINE Offset,PR[78:Offst_apprch]  ;
1511: WAIT   0.20(sec) ;
1512:L P[1082]  R[157] mm/sec CNT100 TA    0.00sec,CALL RUN_LASER_START Offset,PR[25:Start_Offset] ;
1514:L P[1083]  R[157] mm/sec CNT100 Offset,PR[24:Rotate_Offset] ;
1515:L P[1084]  R[157] mm/sec CNT100 TA    0.00sec,CALL RUN_LASER_STOP Offset,PR[26:Stop_Offset] ;
1517:L P[1084]  R[157] mm/sec FINE Offset,PR[76:Offst_dprt] ;
1518:L P[1085]  R[157] mm/sec CNT100 Offset,PR[24:Rotate_Offset] ;
1519:L P[1086]  R[157] mm/sec CNT100 Offset,PR[24:Rotate_Offset] ;
1520:L P[1087]  R[157] mm/sec CNT100 Offset,PR[24:Rotate_Offset] ;
1521:L P[1088]  R[157] mm/sec CNT100 Offset,PR[24:Rotate_Offset] ;
1522:L P[1089]  R[157] mm/sec CNT100 Offset,PR[24:Rotate_Offset] ;
1523:L P[1090]  R[157] mm/sec CNT100 Offset,PR[24:Rotate_Offset] ;
1524: !Pass61 ;
1525: LBL[161:Pass61] ;
1526:L P[1091]  R[157] mm/sec FINE Offset,PR[78:Offst_apprch]  ;
1527: WAIT   0.20(sec) ;
1528:L P[1091]  R[157] mm/sec CNT100 TA    0.00sec,CALL RUN_LASER_START Offset,PR[25:Start_Offset] ;
1530:L P[1092]  R[157] mm/sec CNT100 Offset,PR[24:Rotate_Offset] ;
1531:L P[1093]  R[157] mm/sec CNT100 TA    0.00sec,CALL RUN_LASER_STOP Offset,PR[26:Stop_Offset] ;
1533:L P[1093]  R[157] mm/sec FINE Offset,PR[76:Offst_dprt] ;
1534:L P[1094]  R[157] mm/sec CNT100 Offset,PR[24:Rotate_Offset] ;
1535:L P[1095]  R[157] mm/sec CNT100 Offset,PR[24:Rotate_Offset] ;
1536:L P[1096]  R[157] mm/sec CNT100 Offset,PR[24:Rotate_Offset] ;
1537:L P[1097]  R[157] mm/sec CNT100 Offset,PR[24:Rotate_Offset] ;
1538:L P[1098]  R[157] mm/sec CNT100 Offset,PR[24:Rotate_Offset] ;
1539:L P[1099]  R[157] mm/sec CNT100 Offset,PR[24:Rotate_Offset] ;
1540: !Pass62 ;
1541: LBL[162:Pass62] ;
1542:L P[1100]  R[157] mm/sec FINE Offset,PR[78:Offst_apprch]  ;
1543: WAIT   0.20(sec) ;
1544:L P[1100]  R[157] mm/sec CNT100 TA    0.00sec,CALL RUN_LASER_START Offset,PR[25:Start_Offset] ;
1546:L P[1101]  R[157] mm/sec CNT100 Offset,PR[24:Rotate_Offset] ;
1547:L P[1102]  R[157] mm/sec CNT100 TA    0.00sec,CALL RUN_LASER_STOP Offset,PR[26:Stop_Offset] ;
1549:L P[1102]  R[157] mm/sec FINE Offset,PR[76:Offst_dprt] ;
1550:L P[1103]  R[157] mm/sec CNT100 Offset,PR[24:Rotate_Offset] ;
1551:L P[1104]  R[157] mm/sec CNT100 Offset,PR[24:Rotate_Offset] ;
1552:L P[1105]  R[157] mm/sec CNT100 Offset,PR[24:Rotate_Offset] ;
1553:L P[1106]  R[157] mm/sec CNT100 Offset,PR[24:Rotate_Offset] ;
1554:L P[1107]  R[157] mm/sec CNT100 Offset,PR[24:Rotate_Offset] ;
1555:L P[1108]  R[157] mm/sec CNT100 Offset,PR[24:Rotate_Offset] ;
1556: !Pass63 ;
1557: LBL[163:Pass63] ;
1558:L P[1109]  R[157] mm/sec FINE Offset,PR[78:Offst_apprch]  ;
1559: WAIT   0.20(sec) ;
1560:L P[1109]  R[157] mm/sec CNT100 TA    0.00sec,CALL RUN_LASER_START Offset,PR[25:Start_Offset] ;
1562:L P[1110]  R[157] mm/sec CNT100 Offset,PR[24:Rotate_Offset] ;
1563:L P[1111]  R[157] mm/sec CNT100 TA    0.00sec,CALL RUN_LASER_STOP Offset,PR[26:Stop_Offset] ;
1565:L P[1111]  R[157] mm/sec FINE Offset,PR[76:Offst_dprt] ;
1566:L P[1112]  R[157] mm/sec CNT100 Offset,PR[24:Rotate_Offset] ;
1567:L P[1113]  R[157] mm/sec CNT100 Offset,PR[24:Rotate_Offset] ;
1568:L P[1114]  R[157] mm/sec CNT100 Offset,PR[24:Rotate_Offset] ;
1569:L P[1115]  R[157] mm/sec CNT100 Offset,PR[24:Rotate_Offset] ;
1570:L P[1116]  R[157] mm/sec CNT100 Offset,PR[24:Rotate_Offset] ;
1571:L P[1117]  R[157] mm/sec CNT100 Offset,PR[24:Rotate_Offset] ;
1572: !Pass64 ;
1573: LBL[164:Pass64] ;
1574:L P[1118]  R[157] mm/sec FINE Offset,PR[78:Offst_apprch]  ;
1575: WAIT   0.20(sec) ;
1576:L P[1118]  R[157] mm/sec CNT100 TA    0.00sec,CALL RUN_LASER_START Offset,PR[25:Start_Offset] ;
1578:L P[1119]  R[157] mm/sec CNT100 Offset,PR[24:Rotate_Offset] ;
1579:L P[1120]  R[157] mm/sec CNT100 Offset,PR[24:Rotate_Offset] ;
1580:L P[1121]  R[157] mm/sec CNT100 Offset,PR[24:Rotate_Offset] ;
1581:L P[1122]  R[157] mm/sec CNT100 Offset,PR[24:Rotate_Offset] ;
1582:L P[1123]  R[157] mm/sec CNT100 Offset,PR[24:Rotate_Offset] ;
1583:L P[1124]  R[157] mm/sec CNT100 TA    0.00sec,CALL RUN_LASER_STOP Offset,PR[26:Stop_Offset] ;
1585:L P[1124]  R[157] mm/sec FINE Offset,PR[76:Offst_dprt] ;
1586:L P[1125]  R[157] mm/sec CNT100 Offset,PR[24:Rotate_Offset] ;
1587:L P[1126]  R[157] mm/sec CNT100 Offset,PR[24:Rotate_Offset] ;
1588:L P[1127]  R[157] mm/sec CNT100 Offset,PR[24:Rotate_Offset] ;
1589:L P[1128]  R[157] mm/sec CNT100 Offset,PR[24:Rotate_Offset] ;
1590:L P[1129]  R[157] mm/sec CNT100 Offset,PR[24:Rotate_Offset] ;
1591:L P[1130]  R[157] mm/sec CNT100 Offset,PR[24:Rotate_Offset] ;
1592: !Pass65 ;
1593: LBL[165:Pass65] ;
1594:L P[1131]  R[157] mm/sec FINE Offset,PR[78:Offst_apprch]  ;
1595: WAIT   0.20(sec) ;
1596:L P[1131]  R[157] mm/sec CNT100 TA    0.00sec,CALL RUN_LASER_START Offset,PR[25:Start_Offset] ;
1598:L P[1132]  R[157] mm/sec CNT100 Offset,PR[24:Rotate_Offset] ;
1599:L P[1133]  R[157] mm/sec CNT100 Offset,PR[24:Rotate_Offset] ;
1600:L P[1134]  R[157] mm/sec CNT100 Offset,PR[24:Rotate_Offset] ;
1601:L P[1135]  R[157] mm/sec CNT100 TA    0.00sec,CALL RUN_LASER_STOP Offset,PR[26:Stop_Offset] ;
1603:L P[1135]  R[157] mm/sec FINE Offset,PR[76:Offst_dprt] ;
1604:L P[1136]  R[157] mm/sec CNT100 Offset,PR[24:Rotate_Offset] ;
1605:L P[1137]  R[157] mm/sec CNT100 Offset,PR[24:Rotate_Offset] ;
1606:L P[1138]  R[157] mm/sec CNT100 Offset,PR[24:Rotate_Offset] ;
1607:L P[1139]  R[157] mm/sec CNT100 Offset,PR[24:Rotate_Offset] ;
1608:L P[1140]  R[157] mm/sec CNT100 Offset,PR[24:Rotate_Offset] ;
1609:L P[1141]  R[157] mm/sec CNT100 Offset,PR[24:Rotate_Offset] ;
1610: !Pass66 ;
1611: LBL[166:Pass66] ;
1612:L P[1142]  R[157] mm/sec FINE Offset,PR[78:Offst_apprch]  ;
1613: WAIT   0.20(sec) ;
1614:L P[1142]  R[157] mm/sec CNT100 TA    0.00sec,CALL RUN_LASER_START Offset,PR[25:Start_Offset] ;
1616:L P[1143]  R[157] mm/sec CNT100 Offset,PR[24:Rotate_Offset] ;
1617:L P[1144]  R[157] mm/sec CNT100 Offset,PR[24:Rotate_Offset] ;
1618:L P[1145]  R[157] mm/sec CNT100 Offset,PR[24:Rotate_Offset] ;
1619:L P[1146]  R[157] mm/sec CNT100 TA    0.00sec,CALL RUN_LASER_STOP Offset,PR[26:Stop_Offset] ;
1621:L P[1146]  R[157] mm/sec FINE Offset,PR[76:Offst_dprt] ;
1622:L P[1147]  R[157] mm/sec CNT100 Offset,PR[24:Rotate_Offset] ;
1623:L P[1148]  R[157] mm/sec CNT100 Offset,PR[24:Rotate_Offset] ;
1624:L P[1149]  R[157] mm/sec CNT100 Offset,PR[24:Rotate_Offset] ;
1625:L P[1150]  R[157] mm/sec CNT100 Offset,PR[24:Rotate_Offset] ;
1626:L P[1151]  R[157] mm/sec CNT100 Offset,PR[24:Rotate_Offset] ;
1627:L P[1152]  R[157] mm/sec CNT100 Offset,PR[24:Rotate_Offset] ;
1628: !Pass67 ;
1629: LBL[167:Pass67] ;
1630:L P[1153]  R[157] mm/sec FINE Offset,PR[78:Offst_apprch]  ;
1631: WAIT   0.20(sec) ;
1632:L P[1153]  R[157] mm/sec CNT100 TA    0.00sec,CALL RUN_LASER_START Offset,PR[25:Start_Offset] ;
1634:L P[1154]  R[157] mm/sec CNT100 Offset,PR[24:Rotate_Offset] ;
1635:L P[1155]  R[157] mm/sec CNT100 Offset,PR[24:Rotate_Offset] ;
1636:L P[1156]  R[157] mm/sec CNT100 TA    0.00sec,CALL RUN_LASER_STOP Offset,PR[26:Stop_Offset] ;
1638:L P[1156]  R[157] mm/sec FINE Offset,PR[76:Offst_dprt] ;
1639:L P[1157]  R[157] mm/sec CNT100 Offset,PR[24:Rotate_Offset] ;
1640:L P[1158]  R[157] mm/sec CNT100 Offset,PR[24:Rotate_Offset] ;
1641:L P[1159]  R[157] mm/sec CNT100 Offset,PR[24:Rotate_Offset] ;
1642:L P[1160]  R[157] mm/sec CNT100 Offset,PR[24:Rotate_Offset] ;
1643:L P[1161]  R[157] mm/sec CNT100 Offset,PR[24:Rotate_Offset] ;
1644:L P[1162]  R[157] mm/sec CNT100 Offset,PR[24:Rotate_Offset] ;
1645: !Pass68 ;
1646: LBL[168:Pass68] ;
1647:L P[1163]  R[157] mm/sec FINE Offset,PR[78:Offst_apprch]  ;
1648: WAIT   0.20(sec) ;
1649:L P[1163]  R[157] mm/sec CNT100 TA    0.00sec,CALL RUN_LASER_START Offset,PR[25:Start_Offset] ;
1651:L P[1164]  R[157] mm/sec CNT100 Offset,PR[24:Rotate_Offset] ;
1652:L P[1165]  R[157] mm/sec CNT100 TA    0.00sec,CALL RUN_LASER_STOP Offset,PR[26:Stop_Offset] ;
1654:L P[1165]  R[157] mm/sec FINE Offset,PR[76:Offst_dprt] ;
1655:L P[1166]  R[157] mm/sec CNT100 Offset,PR[24:Rotate_Offset] ;
1656:L P[1167]  R[157] mm/sec CNT100 Offset,PR[24:Rotate_Offset] ;
1657:L P[1168]  R[157] mm/sec CNT100 Offset,PR[24:Rotate_Offset] ;
1658:L P[1169]  R[157] mm/sec CNT100 Offset,PR[24:Rotate_Offset] ;
1659:L P[1170]  R[157] mm/sec CNT100 Offset,PR[24:Rotate_Offset] ;
1660:L P[1171]  R[157] mm/sec CNT100 Offset,PR[24:Rotate_Offset] ;
1661: !Pass69 ;
1662: LBL[169:Pass69] ;
1663:L P[1172]  R[157] mm/sec FINE Offset,PR[78:Offst_apprch]  ;
1664: WAIT   0.20(sec) ;
1665:L P[1172]  R[157] mm/sec CNT100 TA    0.00sec,CALL RUN_LASER_START Offset,PR[25:Start_Offset] ;
1667:L P[1173]  R[157] mm/sec CNT100 Offset,PR[24:Rotate_Offset] ;
1668:L P[1174]  R[157] mm/sec CNT100 Offset,PR[24:Rotate_Offset] ;
1669:L P[1175]  R[157] mm/sec CNT100 Offset,PR[24:Rotate_Offset] ;
1670:L P[1176]  R[157] mm/sec CNT100 TA    0.00sec,CALL RUN_LASER_STOP Offset,PR[26:Stop_Offset] ;
1672:L P[1176]  R[157] mm/sec FINE Offset,PR[76:Offst_dprt] ;
1673:L P[1177]  R[157] mm/sec CNT100 Offset,PR[24:Rotate_Offset] ;
1674:L P[1178]  R[157] mm/sec CNT100 Offset,PR[24:Rotate_Offset] ;
1675:L P[1179]  R[157] mm/sec CNT100 Offset,PR[24:Rotate_Offset] ;
1676:L P[1180]  R[157] mm/sec CNT100 Offset,PR[24:Rotate_Offset] ;
1677:L P[1181]  R[157] mm/sec CNT100 Offset,PR[24:Rotate_Offset] ;
1678:L P[1182]  R[157] mm/sec CNT100 Offset,PR[24:Rotate_Offset] ;
1679: !Pass70 ;
1680: LBL[170:Pass70] ;
1681:L P[1183]  R[157] mm/sec FINE Offset,PR[78:Offst_apprch]  ;
1682: WAIT   0.20(sec) ;
1683:L P[1183]  R[157] mm/sec CNT100 TA    0.00sec,CALL RUN_LASER_START Offset,PR[25:Start_Offset] ;
1685:L P[1184]  R[157] mm/sec CNT100 Offset,PR[24:Rotate_Offset] ;
1686:L P[1185]  R[157] mm/sec CNT100 Offset,PR[24:Rotate_Offset] ;
1687:L P[1186]  R[157] mm/sec CNT100 TA    0.00sec,CALL RUN_LASER_STOP Offset,PR[26:Stop_Offset] ;
1689:L P[1186]  R[157] mm/sec FINE Offset,PR[76:Offst_dprt] ;
1690:L P[1187]  R[157] mm/sec CNT100 Offset,PR[24:Rotate_Offset] ;
1691:L P[1188]  R[157] mm/sec CNT100 Offset,PR[24:Rotate_Offset] ;
1692:L P[1189]  R[157] mm/sec CNT100 Offset,PR[24:Rotate_Offset] ;
1693:L P[1190]  R[157] mm/sec CNT100 Offset,PR[24:Rotate_Offset] ;
1694:L P[1191]  R[157] mm/sec CNT100 Offset,PR[24:Rotate_Offset] ;
1695:L P[1192]  R[157] mm/sec CNT100 Offset,PR[24:Rotate_Offset] ;
1696: !Pass71 ;
1697: LBL[171:Pass71] ;
1698:L P[1193]  R[157] mm/sec FINE Offset,PR[78:Offst_apprch]  ;
1699: WAIT   0.20(sec) ;
1700:L P[1193]  R[157] mm/sec CNT100 TA    0.00sec,CALL RUN_LASER_START Offset,PR[25:Start_Offset] ;
1702:L P[1194]  R[157] mm/sec CNT100 Offset,PR[24:Rotate_Offset] ;
1703:L P[1195]  R[157] mm/sec CNT100 Offset,PR[24:Rotate_Offset] ;
1704:L P[1196]  R[157] mm/sec CNT100 Offset,PR[24:Rotate_Offset] ;
1705:L P[1197]  R[157] mm/sec CNT100 Offset,PR[24:Rotate_Offset] ;
1706:L P[1198]  R[157] mm/sec CNT100 Offset,PR[24:Rotate_Offset] ;
1707:L P[1199]  R[157] mm/sec CNT100 TA    0.00sec,CALL RUN_LASER_STOP Offset,PR[26:Stop_Offset] ;
1709:L P[1199]  R[157] mm/sec FINE Offset,PR[76:Offst_dprt] ;
1710:L P[1200]  R[157] mm/sec CNT100 Offset,PR[24:Rotate_Offset] ;
1711:L P[1201]  R[157] mm/sec CNT100 Offset,PR[24:Rotate_Offset] ;
1712:L P[1202]  R[157] mm/sec CNT100 Offset,PR[24:Rotate_Offset] ;
1713:L P[1203]  R[157] mm/sec CNT100 Offset,PR[24:Rotate_Offset] ;
1714:L P[1204]  R[157] mm/sec CNT100 Offset,PR[24:Rotate_Offset] ;
1715:L P[1205]  R[157] mm/sec CNT100 Offset,PR[24:Rotate_Offset] ;
1716: !Pass72 ;
1717: LBL[172:Pass72] ;
1718:L P[1206]  R[157] mm/sec FINE Offset,PR[78:Offst_apprch]  ;
1719: WAIT   0.20(sec) ;
1720:L P[1206]  R[157] mm/sec CNT100 TA    0.00sec,CALL RUN_LASER_START Offset,PR[25:Start_Offset] ;
1722:L P[1207]  R[157] mm/sec CNT100 Offset,PR[24:Rotate_Offset] ;
1723:L P[1208]  R[157] mm/sec CNT100 TA    0.00sec,CALL RUN_LASER_STOP Offset,PR[26:Stop_Offset] ;
1725:L P[1208]  R[157] mm/sec FINE Offset,PR[76:Offst_dprt] ;
1726:L P[1209]  R[157] mm/sec CNT100 Offset,PR[24:Rotate_Offset] ;
1727:L P[1210]  R[157] mm/sec CNT100 Offset,PR[24:Rotate_Offset] ;
1728:L P[1211]  R[157] mm/sec CNT100 Offset,PR[24:Rotate_Offset] ;
1729:L P[1212]  R[157] mm/sec CNT100 Offset,PR[24:Rotate_Offset] ;
1730:L P[1213]  R[157] mm/sec CNT100 Offset,PR[24:Rotate_Offset] ;
1731:L P[1214]  R[157] mm/sec CNT100 Offset,PR[24:Rotate_Offset] ;
1732: !Pass73 ;
1733: LBL[173:Pass73] ;
1734:L P[1215]  R[157] mm/sec FINE Offset,PR[78:Offst_apprch]  ;
1735: WAIT   0.20(sec) ;
1736:L P[1215]  R[157] mm/sec CNT100 TA    0.00sec,CALL RUN_LASER_START Offset,PR[25:Start_Offset] ;
1738:L P[1216]  R[157] mm/sec CNT100 Offset,PR[24:Rotate_Offset] ;
1739:L P[1217]  R[157] mm/sec CNT100 TA    0.00sec,CALL RUN_LASER_STOP Offset,PR[26:Stop_Offset] ;
1741:L P[1217]  R[157] mm/sec FINE Offset,PR[76:Offst_dprt] ;
